   1:  PR[91,2] = PR[90,2] + -8.319;
   1:  PR[91,3] = PR[90,3] + 6.919;
   1:L PR[91] R[100]mm/sec CNT100;
   1:  PR[91,1] = PR[90,1] + 34.688;
   1:  PR[91,2] = PR[90,2] + -7.593;
   1:  PR[91,3] = PR[90,3] + 6.924;
   1:L PR[91] R[100]mm/sec CNT100;
   1:  PR[91,1] = PR[90,1] + 35.067;
   1:  PR[91,2] = PR[90,2] + -6.848;
   1:  PR[91,3] = PR[90,3] + 6.929;
   1:L PR[91] R[100]mm/sec CNT100;
   1:  PR[91,1] = PR[90,1] + 35.409;
   1:  PR[91,2] = PR[90,2] + -6.085;
   1:  PR[91,3] = PR[90,3] + 6.934;
   1:L PR[91] R[100]mm/sec CNT100;
   1:  PR[91,1] = PR[90,1] + 35.712;
   1:  PR[91,2] = PR[90,2] + -5.307;
   1:  PR[91,3] = PR[90,3] + 6.939;
   1:L PR[91] R[100]mm/sec CNT100;
   1:  PR[91,1] = PR[90,1] + 35.976;
   1:  PR[91,2] = PR[90,2] + -4.515;
   1:  PR[91,3] = PR[90,3] + 6.944;
   1:L PR[91] R[100]mm/sec CNT100;
   1:  PR[91,1] = PR[90,1] + 36.201;
   1:  PR[91,2] = PR[90,2] + -3.712;
   1:  PR[91,3] = PR[90,3] + 6.950;
   1:L PR[91] R[100]mm/sec CNT100;
   1:  PR[91,1] = PR[90,1] + 36.386;
   1:  PR[91,2] = PR[90,2] + -2.898;
   1:  PR[91,3] = PR[90,3] + 6.955;
   1:L PR[91] R[100]mm/sec CNT100;
   1:  PR[91,1] = PR[90,1] + 36.530;
   1:  PR[91,2] = PR[90,2] + -2.076;
   1:  PR[91,3] = PR[90,3] + 6.960;
   1:L PR[91] R[100]mm/sec CNT100;
   1:  PR[91,1] = PR[90,1] + 36.633;
   1:  PR[91,2] = PR[90,2] + -1.246;
   1:  PR[91,3] = PR[90,3] + 6.965;
   1:L PR[91] R[100]mm/sec CNT100;
   1:  PR[91,1] = PR[90,1] + 36.695;
   1:  PR[91,2] = PR[90,2] + -0.411;
   1:  PR[91,3] = PR[90,3] + 6.970;
   1:L PR[91] R[100]mm/sec CNT100;
   1:  PR[91,1] = PR[90,1] + 36.716;
   1:  PR[91,2] = PR[90,2] + 0.428;
   1:  PR[91,3] = PR[90,3] + 6.975;
   1:L PR[91] R[100]mm/sec CNT100;
   1:  PR[91,1] = PR[90,1] + 36.695;
   1:  PR[91,2] = PR[90,2] + 1.266;
   1:  PR[91,3] = PR[90,3] + 6.980;
   1:L PR[91] R[100]mm/sec CNT100;
   1:  PR[91,1] = PR[90,1] + 36.633;
   1:  PR[91,2] = PR[90,2] + 2.101;
   1:  PR[91,3] = PR[90,3] + 6.985;
   1:L PR[91] R[100]mm/sec CNT100;
   1:  PR[91,1] = PR[90,1] + 36.530;
   1:  PR[91,2] = PR[90,2] + 2.931;
   1:  PR[91,3] = PR[90,3] + 6.990;
   1:L PR[91] R[100]mm/sec CNT100;
   1:  PR[91,1] = PR[90,1] + 36.386;
   1:  PR[91,2] = PR[90,2] + 3.753;
   1:  PR[91,3] = PR[90,3] + 6.995;
   1:L PR[91] R[100]mm/sec CNT100;
   1:  PR[91,1] = PR[90,1] + 36.201;
   1:  PR[91,2] = PR[90,2] + 4.567;
   1:  PR[91,3] = PR[90,3] + 7.000;
   1:L PR[91] R[100]mm/sec CNT100;
   1:  PR[91,1] = PR[90,1] + 35.976;
   1:  PR[91,2] = PR[90,2] + 5.371;
   1:  PR[91,3] = PR[90,3] + 7.005;
   1:L PR[91] R[100]mm/sec CNT100;
   1:  PR[91,1] = PR[90,1] + 35.712;
   1:  PR[91,2] = PR[90,2] + 6.162;
   1:  PR[91,3] = PR[90,3] + 7.011;
   1:L PR[91] R[100]mm/sec CNT100;
   1:  PR[91,1] = PR[90,1] + 35.409;
   1:  PR[91,2] = PR[90,2] + 6.940;
   1:  PR[91,3] = PR[90,3] + 7.016;
   1:L PR[91] R[100]mm/sec CNT100;
   1:  PR[91,1] = PR[90,1] + 35.067;
   1:  PR[91,2] = PR[90,2] + 7.703;
   1:  PR[91,3] = PR[90,3] + 7.021;
   1:L PR[91] R[100]mm/sec CNT100;
   1:  PR[91,1] = PR[90,1] + 34.688;
   1:  PR[91,2] = PR[90,2] + 8.449;
   1:  PR[91,3] = PR[90,3] + 7.026;
   1:L PR[91] R[100]mm/sec CNT100;
   1:  PR[91,1] = PR[90,1] + 34.273;
   1:  PR[91,2] = PR[90,2] + 9.175;
   1:  PR[91,3] = PR[90,3] + 7.031;
   1:L PR[91] R[100]mm/sec CNT100;
   1:  PR[91,1] = PR[90,1] + 33.822;
   1:  PR[91,2] = PR[90,2] + 9.879;
   1:  PR[91,3] = PR[90,3] + 7.036;
   1:L PR[91] R[100]mm/sec CNT100;
   1:  PR[91,1] = PR[90,1] + 33.337;
   1:  PR[91,2] = PR[90,2] + 10.561;
   1:  PR[91,3] = PR[90,3] + 7.041;
   1:L PR[91] R[100]mm/sec CNT100;
   1:  PR[91,1] = PR[90,1] + 32.819;
   1:  PR[91,2] = PR[90,2] + 11.219;
   1:  PR[91,3] = PR[90,3] + 7.046;
   1:L PR[91] R[100]mm/sec CNT100;
   1:  PR[91,1] = PR[90,1] + 32.269;
   1:  PR[91,2] = PR[90,2] + 11.849;
   1:  PR[91,3] = PR[90,3] + 7.051;
   1:L PR[91] R[100]mm/sec CNT100;
   1:  PR[91,1] = PR[90,1] + 31.688;
   1:  PR[91,2] = PR[90,2] + 12.452;
   1:  PR[91,3] = PR[90,3] + 7.056;
   1:L PR[91] R[100]mm/sec CNT100;
   1:  PR[91,1] = PR[90,1] + 31.079;
   1:  PR[91,2] = PR[90,2] + 13.025;
   1:  PR[91,3] = PR[90,3] + 7.061;
   1:L PR[91] R[100]mm/sec CNT100;
   1:  PR[91,1] = PR[90,1] + 30.441;
   1:  PR[91,2] = PR[90,2] + 13.567;
   1:  PR[91,3] = PR[90,3] + 7.067;
   1:L PR[91] R[100]mm/sec CNT100;
   1:  PR[91,1] = PR[90,1] + 29.778;
   1:  PR[91,2] = PR[90,2] + 14.078;
   1:  PR[91,3] = PR[90,3] + 7.072;
   1:L PR[91] R[100]mm/sec CNT100;
   1:  PR[91,1] = PR[90,1] + 29.090;
   1:  PR[91,2] = PR[90,2] + 14.555;
   1:  PR[91,3] = PR[90,3] + 7.077;
   1:L PR[91] R[100]mm/sec CNT100;
   1:  PR[91,1] = PR[90,1] + 28.379;
   1:  PR[91,2] = PR[90,2] + 14.998;
   1:  PR[91,3] = PR[90,3] + 7.082;
   1:L PR[91] R[100]mm/sec CNT100;
   1:  PR[91,1] = PR[90,1] + 27.647;
   1:  PR[91,2] = PR[90,2] + 15.405;
   1:  PR[91,3] = PR[90,3] + 7.087;
   1:L PR[91] R[100]mm/sec CNT100;
   1:  PR[91,1] = PR[90,1] + 26.895;
   1:  PR[91,2] = PR[90,2] + 15.775;
   1:  PR[91,3] = PR[90,3] + 7.092;
   1:L PR[91] R[100]mm/sec CNT100;
   1:  PR[91,1] = PR[90,1] + 26.126;
   1:  PR[91,2] = PR[90,2] + 16.108;
   1:  PR[91,3] = PR[90,3] + 7.097;
   1:L PR[91] R[100]mm/sec CNT100;
   1:  PR[91,1] = PR[90,1] + 25.342;
   1:  PR[91,2] = PR[90,2] + 16.403;
   1:  PR[91,3] = PR[90,3] + 7.102;
   1:L PR[91] R[100]mm/sec CNT100;
   1:  PR[91,1] = PR[90,1] + 24.544;
   1:  PR[91,2] = PR[90,2] + 16.659;
   1:  PR[91,3] = PR[90,3] + 7.107;
   1:L PR[91] R[100]mm/sec CNT100;
   1:  PR[91,1] = PR[90,1] + 23.734;
   1:  PR[91,2] = PR[90,2] + 16.875;
   1:  PR[91,3] = PR[90,3] + 7.112;
   1:L PR[91] R[100]mm/sec CNT100;
   1:  PR[91,1] = PR[90,1] + 22.914;
   1:  PR[91,2] = PR[90,2] + 17.051;
   1:  PR[91,3] = PR[90,3] + 7.117;
   1:L PR[91] R[100]mm/sec CNT100;
   1:  PR[91,1] = PR[90,1] + 22.086;
   1:  PR[91,2] = PR[90,2] + 17.187;
   1:  PR[91,3] = PR[90,3] + 7.123;
   1:L PR[91] R[100]mm/sec CNT100;
   1:  PR[91,1] = PR[90,1] + 21.253;
   1:  PR[91,2] = PR[90,2] + 17.281;
   1:  PR[91,3] = PR[90,3] + 7.128;
   1:L PR[91] R[100]mm/sec CNT100;
   1:  PR[91,1] = PR[90,1] + 20.416;
   1:  PR[91,2] = PR[90,2] + 17.335;
   1:  PR[91,3] = PR[90,3] + 7.133;
   1:L PR[91] R[100]mm/sec CNT100;
   1:  PR[91,1] = PR[90,1] + 19.577;
   1:  PR[91,2] = PR[90,2] + 17.347;
   1:  PR[91,3] = PR[90,3] + 7.138;
   1:L PR[91] R[100]mm/sec CNT100;
   1:  PR[91,1] = PR[90,1] + 18.739;
   1:  PR[91,2] = PR[90,2] + 17.318;
   1:  PR[91,3] = PR[90,3] + 7.143;
   1:L PR[91] R[100]mm/sec CNT100;
   1:  PR[91,1] = PR[90,1] + 17.902;
   1:  PR[91,2] = PR[90,2] + 17.247;
   1:  PR[91,3] = PR[90,3] + 7.148;
   1:L PR[91] R[100]mm/sec CNT100;
   1:  PR[91,1] = PR[90,1] + 17.071;
   1:  PR[91,2] = PR[90,2] + 17.136;
   1:  PR[91,3] = PR[90,3] + 7.153;
   1:L PR[91] R[100]mm/sec CNT100;
   1:  PR[91,1] = PR[90,1] + 16.226;
   1:  PR[91,2] = PR[90,2] + 16.978;
   1:  PR[91,3] = PR[90,3] + 7.158;
   1:L PR[91] R[100]mm/sec CNT100;
   1:  PR[91,1] = PR[90,1] + 15.428;
   1:  PR[91,2] = PR[90,2] + 16.790;
   1:  PR[91,3] = PR[90,3] + 7.164;
   1:L PR[91] R[100]mm/sec CNT100;
   1:  PR[91,1] = PR[90,1] + 14.620;
   1:  PR[91,2] = PR[90,2] + 16.557;
   1:  PR[91,3] = PR[90,3] + 7.168;
   1:L PR[91] R[100]mm/sec CNT100;
   1:  PR[91,1] = PR[90,1] + 13.825;
   1:  PR[91,2] = PR[90,2] + 16.285;
   1:  PR[91,3] = PR[90,3] + 7.174;
   1:L PR[91] R[100]mm/sec CNT100;
   1:  PR[91,1] = PR[90,1] + 13.044;
   1:  PR[91,2] = PR[90,2] + 15.974;
   1:  PR[91,3] = PR[90,3] + 7.179;
   1:L PR[91] R[100]mm/sec CNT100;
   1:  PR[91,1] = PR[90,1] + 12.279;
   1:  PR[91,2] = PR[90,2] + 15.624;
   1:  PR[91,3] = PR[90,3] + 7.184;
   1:L PR[91] R[100]mm/sec CNT100;
   1:  PR[91,1] = PR[90,1] + 11.533;
   1:  PR[91,2] = PR[90,2] + 15.238;
   1:  PR[91,3] = PR[90,3] + 7.189;
   1:L PR[91] R[100]mm/sec CNT100;
   1:  PR[91,1] = PR[90,1] + 10.807;
   1:  PR[91,2] = PR[90,2] + 14.816;
   1:  PR[91,3] = PR[90,3] + 7.194;
   1:L PR[91] R[100]mm/sec CNT100;
   1:  PR[91,1] = PR[90,1] + 10.102;
   1:  PR[91,2] = PR[90,2] + 14.358;
   1:  PR[91,3] = PR[90,3] + 7.199;
   1:L PR[91] R[100]mm/sec CNT100;
   1:  PR[91,1] = PR[90,1] + 9.421;
   1:  PR[91,2] = PR[90,2] + 13.866;
   1:  PR[91,3] = PR[90,3] + 7.204;
   1:L PR[91] R[100]mm/sec CNT100;
   1:  PR[91,1] = PR[90,1] + 8.765;
   1:  PR[91,2] = PR[90,2] + 13.341;
   1:  PR[91,3] = PR[90,3] + 7.209;
   1:L PR[91] R[100]mm/sec CNT100;
   1:  PR[91,1] = PR[90,1] + 8.136;
   1:  PR[91,2] = PR[90,2] + 12.785;
   1:  PR[91,3] = PR[90,3] + 7.214;
   1:L PR[91] R[100]mm/sec CNT100;
   1:  PR[91,1] = PR[90,1] + 7.535;
   1:  PR[91,2] = PR[90,2] + 12.198;
   1:  PR[91,3] = PR[90,3] + 7.220;
   1:L PR[91] R[100]mm/sec CNT100;
   1:  PR[91,1] = PR[90,1] + 6.965;
   1:  PR[91,2] = PR[90,2] + 11.581;
   1:  PR[91,3] = PR[90,3] + 7.225;
   1:L PR[91] R[100]mm/sec CNT100;
   1:  PR[91,1] = PR[90,1] + 6.425;
   1:  PR[91,2] = PR[90,2] + 10.938;
   1:  PR[91,3] = PR[90,3] + 7.230;
   1:L PR[91] R[100]mm/sec CNT100;
   1:  PR[91,1] = PR[90,1] + 5.918;
   1:  PR[91,2] = PR[90,2] + 10.268;
   1:  PR[91,3] = PR[90,3] + 7.235;
   1:L PR[91] R[100]mm/sec CNT100;
   1:  PR[91,1] = PR[90,1] + 5.445;
   1:  PR[91,2] = PR[90,2] + 9.574;
   1:  PR[91,3] = PR[90,3] + 7.240;
   1:L PR[91] R[100]mm/sec CNT100;
   1:  PR[91,1] = PR[90,1] + 5.007;
   1:  PR[91,2] = PR[90,2] + 8.857;
   1:  PR[91,3] = PR[90,3] + 7.245;
   1:L PR[91] R[100]mm/sec CNT100;
   1:  PR[91,1] = PR[90,1] + 4.605;
   1:  PR[91,2] = PR[90,2] + 8.120;
   1:  PR[91,3] = PR[90,3] + 7.250;
   1:L PR[91] R[100]mm/sec CNT100;
   1:  PR[91,1] = PR[90,1] + 4.240;
   1:  PR[91,2] = PR[90,2] + 7.365;
   1:  PR[91,3] = PR[90,3] + 7.255;
   1:L PR[91] R[100]mm/sec CNT100;
   1:  PR[91,1] = PR[90,1] + 3.913;
   1:  PR[91,2] = PR[90,2] + 6.594;
   1:  PR[91,3] = PR[90,3] + 7.260;
   1:L PR[91] R[100]mm/sec CNT100;
   1:  PR[91,1] = PR[90,1] + 3.625;
   1:  PR[91,2] = PR[90,2] + 5.810;
   1:  PR[91,3] = PR[90,3] + 7.266;
   1:L PR[91] R[100]mm/sec CNT100;
   1:  PR[91,1] = PR[90,1] + 3.377;
   1:  PR[91,2] = PR[90,2] + 5.013;
   1:  PR[91,3] = PR[90,3] + 7.271;
   1:L PR[91] R[100]mm/sec CNT100;
   1:  PR[91,1] = PR[90,1] + 3.169;
   1:  PR[91,2] = PR[90,2] + 4.205;
   1:  PR[91,3] = PR[90,3] + 7.276;
   1:L PR[91] R[100]mm/sec CNT100;
   1:  PR[91,1] = PR[90,1] + 2.997;
   1:  PR[91,2] = PR[90,2] + 3.358;
   1:  PR[91,3] = PR[90,3] + 7.281;
   1:L PR[91] R[100]mm/sec CNT100;
   1:  PR[91,1] = PR[90,1] + 2.902;
   1:  PR[91,2] = PR[90,2] + 2.988;
   1:  PR[91,3] = PR[90,3] + 7.286;
   1:L PR[91] R[100]mm/sec CNT100;
   1:  PR[91,1] = PR[90,1] + 2.754;
   1:  PR[91,2] = PR[90,2] + 2.613;
   1:  PR[91,3] = PR[90,3] + 7.288;
   1:L PR[91] R[100]mm/sec CNT100;
   1:  PR[91,1] = PR[90,1] + 2.570;
   1:  PR[91,2] = PR[90,2] + 2.280;
   1:  PR[91,3] = PR[90,3] + 7.291;
   1:L PR[91] R[100]mm/sec CNT100;
   1:  PR[91,1] = PR[90,1] + 2.373;
   1:  PR[91,2] = PR[90,2] + 2.003;
   1:  PR[91,3] = PR[90,3] + 7.293;
   1:L PR[91] R[100]mm/sec CNT100;
   1:  PR[91,1] = PR[90,1] + 2.094;
   1:  PR[91,2] = PR[90,2] + 1.696;
   1:  PR[91,3] = PR[90,3] + 7.295;
   1:L PR[91] R[100]mm/sec CNT100;
   1:  PR[91,1] = PR[90,1] + 1.771;
   1:  PR[91,2] = PR[90,2] + 1.427;
   1:  PR[91,3] = PR[90,3] + 7.298;
   1:L PR[91] R[100]mm/sec CNT100;
   1:  PR[91,1] = PR[90,1] + 1.413;
   1:  PR[91,2] = PR[90,2] + 1.202;
   1:  PR[91,3] = PR[90,3] + 7.300;
   1:L PR[91] R[100]mm/sec CNT100;
   1:  PR[91,1] = PR[90,1] + 1.037;
   1:  PR[91,2] = PR[90,2] + 1.031;
   1:  PR[91,3] = PR[90,3] + 7.303;
   1:L PR[91] R[100]mm/sec CNT100;
   1:  PR[91,1] = PR[90,1] + 0.744;
   1:  PR[91,2] = PR[90,2] + 0.936;
   1:  PR[91,3] = PR[90,3] + 7.305;
   1:L PR[91] R[100]mm/sec CNT100;
   1:  PR[91,1] = PR[90,1] + 0.340;
   1:  PR[91,2] = PR[90,2] + 0.854;
   1:  PR[91,3] = PR[90,3] + 7.307;
   1:L PR[91] R[100]mm/sec CNT100;
   1:  PR[91,1] = PR[90,1] + -0.072;
   1:  PR[91,2] = PR[90,2] + 0.827;
   1:  PR[91,3] = PR[90,3] + 7.310;
   1:L PR[91] R[100]mm/sec CNT100;
   1:  PR[91,1] = PR[90,1] + -0.523;
   1:  PR[91,2] = PR[90,2] + 0.847;
   1:  PR[91,3] = PR[90,3] + 7.312;
   1:L PR[91] R[100]mm/sec CNT100;
   1:  PR[91,1] = PR[90,1] + -0.953;
   1:  PR[91,2] = PR[90,2] + 0.928;
   1:  PR[91,3] = PR[90,3] + 7.315;
   1:L PR[91] R[100]mm/sec CNT100;
   1:  PR[91,1] = PR[90,1] + -1.273;
   1:  PR[91,2] = PR[90,2] + 1.030;
   1:  PR[91,3] = PR[90,3] + 7.318;
   1:L PR[91] R[100]mm/sec CNT100;
   1:  PR[91,1] = PR[90,1] + -1.637;
   1:  PR[91,2] = PR[90,2] + 1.194;
   1:  PR[91,3] = PR[90,3] + 7.320;
   1:L PR[91] R[100]mm/sec CNT100;
   1:  PR[91,1] = PR[90,1] + -1.982;
   1:  PR[91,2] = PR[90,2] + 1.407;
   1:  PR[91,3] = PR[90,3] + 7.322;
   1:L PR[91] R[100]mm/sec CNT100;
   1:  PR[91,1] = PR[90,1] + -2.261;
   1:  PR[91,2] = PR[90,2] + 1.632;
   1:  PR[91,3] = PR[90,3] + 7.325;
   1:L PR[91] R[100]mm/sec CNT100;
   1:  PR[91,1] = PR[90,1] + -2.628;
   1:  PR[91,2] = PR[90,2] + 2.025;
   1:  PR[91,3] = PR[90,3] + 7.327;
   1:L PR[91] R[100]mm/sec CNT100;
   1:  PR[91,1] = PR[90,1] + -2.823;
   1:  PR[91,2] = PR[90,2] + 2.302;
   1:  PR[91,3] = PR[90,3] + 7.330;
   1:L PR[91] R[100]mm/sec CNT100;
   1:  PR[91,1] = PR[90,1] + -3.001;
   1:  PR[91,2] = PR[90,2] + 2.631;
   1:  PR[91,3] = PR[90,3] + 7.332;
   1:L PR[91] R[100]mm/sec CNT100;
   1:  PR[91,1] = PR[90,1] + -3.158;
   1:  PR[91,2] = PR[90,2] + 3.044;
   1:  PR[91,3] = PR[90,3] + 7.334;
   1:L PR[91] R[100]mm/sec CNT100;
   1:  PR[91,1] = PR[90,1] + -3.406;
   1:  PR[91,2] = PR[90,2] + 4.200;
   1:  PR[91,3] = PR[90,3] + 7.337;
   1:L PR[91] R[100]mm/sec CNT100;
   1:  PR[91,1] = PR[90,1] + -3.615;
   1:  PR[91,2] = PR[90,2] + 5.011;
   1:  PR[91,3] = PR[90,3] + 7.344;
   1:L PR[91] R[100]mm/sec CNT100;
   1:  PR[91,1] = PR[90,1] + -3.864;
   1:  PR[91,2] = PR[90,2] + 5.809;
   1:  PR[91,3] = PR[90,3] + 7.349;
   1:L PR[91] R[100]mm/sec CNT100;
   1:  PR[91,1] = PR[90,1] + -4.152;
   1:  PR[91,2] = PR[90,2] + 6.594;
   1:  PR[91,3] = PR[90,3] + 7.354;
   1:L PR[91] R[100]mm/sec CNT100;
   1:  PR[91,1] = PR[90,1] + -4.479;
   1:  PR[91,2] = PR[90,2] + 7.366;
   1:  PR[91,3] = PR[90,3] + 7.360;
   1:L PR[91] R[100]mm/sec CNT100;
   1:  PR[91,1] = PR[90,1] + -4.844;
   1:  PR[91,2] = PR[90,2] + 8.122;
   1:  PR[91,3] = PR[90,3] + 7.365;
   1:L PR[91] R[100]mm/sec CNT100;
   1:  PR[91,1] = PR[90,1] + -5.246;
   1:  PR[91,2] = PR[90,2] + 8.859;
   1:  PR[91,3] = PR[90,3] + 7.370;
   1:L PR[91] R[100]mm/sec CNT100;
   1:  PR[91,1] = PR[90,1] + -5.684;
   1:  PR[91,2] = PR[90,2] + 9.576;
   1:  PR[91,3] = PR[90,3] + 7.375;
   1:L PR[91] R[100]mm/sec CNT100;
   1:  PR[91,1] = PR[90,1] + -6.157;
   1:  PR[91,2] = PR[90,2] + 10.270;
   1:  PR[91,3] = PR[90,3] + 7.380;
   1:L PR[91] R[100]mm/sec CNT100;
   1:  PR[91,1] = PR[90,1] + -6.664;
   1:  PR[91,2] = PR[90,2] + 10.939;
   1:  PR[91,3] = PR[90,3] + 7.385;
   1:L PR[91] R[100]mm/sec CNT100;
   1:  PR[91,1] = PR[90,1] + -7.204;
   1:  PR[91,2] = PR[90,2] + 11.583;
   1:  PR[91,3] = PR[90,3] + 7.390;
   1:L PR[91] R[100]mm/sec CNT100;
   1:  PR[91,1] = PR[90,1] + -7.775;
   1:  PR[91,2] = PR[90,2] + 12.198;
   1:  PR[91,3] = PR[90,3] + 7.395;
   1:L PR[91] R[100]mm/sec CNT100;
   1:  PR[91,1] = PR[90,1] + -8.375;
   1:  PR[91,2] = PR[90,2] + 12.785;
   1:  PR[91,3] = PR[90,3] + 7.400;
   1:L PR[91] R[100]mm/sec CNT100;
   1:  PR[91,1] = PR[90,1] + -9.004;
   1:  PR[91,2] = PR[90,2] + 13.341;
   1:  PR[91,3] = PR[90,3] + 7.405;
   1:L PR[91] R[100]mm/sec CNT100;
   1:  PR[91,1] = PR[90,1] + -9.660;
   1:  PR[91,2] = PR[90,2] + 13.866;
   1:  PR[91,3] = PR[90,3] + 7.411;
   1:L PR[91] R[100]mm/sec CNT100;
   1:  PR[91,1] = PR[90,1] + -10.341;
   1:  PR[91,2] = PR[90,2] + 14.358;
   1:  PR[91,3] = PR[90,3] + 7.416;
   1:L PR[91] R[100]mm/sec CNT100;
   1:  PR[91,1] = PR[90,1] + -11.046;
   1:  PR[91,2] = PR[90,2] + 14.816;
   1:  PR[91,3] = PR[90,3] + 7.421;
   1:L PR[91] R[100]mm/sec CNT100;
   1:  PR[91,1] = PR[90,1] + -11.772;
   1:  PR[91,2] = PR[90,2] + 15.238;
   1:  PR[91,3] = PR[90,3] + 7.426;
   1:L PR[91] R[100]mm/sec CNT100;
   1:  PR[91,1] = PR[90,1] + -12.519;
   1:  PR[91,2] = PR[90,2] + 15.625;
   1:  PR[91,3] = PR[90,3] + 7.431;
   1:L PR[91] R[100]mm/sec CNT100;
   1:  PR[91,1] = PR[90,1] + -13.283;
   1:  PR[91,2] = PR[90,2] + 15.974;
   1:  PR[91,3] = PR[90,3] + 7.436;
   1:L PR[91] R[100]mm/sec CNT100;
   1:  PR[91,1] = PR[90,1] + -14.064;
   1:  PR[91,2] = PR[90,2] + 16.285;
   1:  PR[91,3] = PR[90,3] + 7.441;
   1:L PR[91] R[100]mm/sec CNT100;
   1:  PR[91,1] = PR[90,1] + -14.859;
   1:  PR[91,2] = PR[90,2] + 16.557;
   1:  PR[91,3] = PR[90,3] + 7.446;
   1:L PR[91] R[100]mm/sec CNT100;
   1:  PR[91,1] = PR[90,1] + -15.678;
   1:  PR[91,2] = PR[90,2] + 16.793;
   1:  PR[91,3] = PR[90,3] + 7.451;
   1:L PR[91] R[100]mm/sec CNT100;
   1:  PR[91,1] = PR[90,1] + -16.484;
   1:  PR[91,2] = PR[90,2] + 16.983;
   1:  PR[91,3] = PR[90,3] + 7.457;
   1:L PR[91] R[100]mm/sec CNT100;
   1:  PR[91,1] = PR[90,1] + -17.310;
   1:  PR[91,2] = PR[90,2] + 17.136;
   1:  PR[91,3] = PR[90,3] + 7.462;
   1:L PR[91] R[100]mm/sec CNT100;
   1:  PR[91,1] = PR[90,1] + -18.141;
   1:  PR[91,2] = PR[90,2] + 17.247;
   1:  PR[91,3] = PR[90,3] + 7.467;
   1:L PR[91] R[100]mm/sec CNT100;
   1:  PR[91,1] = PR[90,1] + -18.978;
   1:  PR[91,2] = PR[90,2] + 17.318;
   1:  PR[91,3] = PR[90,3] + 7.472;
   1:L PR[91] R[100]mm/sec CNT100;
   1:  PR[91,1] = PR[90,1] + -19.816;
   1:  PR[91,2] = PR[90,2] + 17.347;
   1:  PR[91,3] = PR[90,3] + 7.477;
   1:L PR[91] R[100]mm/sec CNT100;
   1:  PR[91,1] = PR[90,1] + -20.655;
   1:  PR[91,2] = PR[90,2] + 17.335;
   1:  PR[91,3] = PR[90,3] + 7.482;
   1:L PR[91] R[100]mm/sec CNT100;
   1:  PR[91,1] = PR[90,1] + -21.492;
   1:  PR[91,2] = PR[90,2] + 17.281;
   1:  PR[91,3] = PR[90,3] + 7.487;
   1:L PR[91] R[100]mm/sec CNT100;
   1:  PR[91,1] = PR[90,1] + -22.325;
   1:  PR[91,2] = PR[90,2] + 17.187;
   1:  PR[91,3] = PR[90,3] + 7.492;
   1:L PR[91] R[100]mm/sec CNT100;
   1:  PR[91,1] = PR[90,1] + -23.153;
   1:  PR[91,2] = PR[90,2] + 17.051;
   1:  PR[91,3] = PR[90,3] + 7.497;
   1:L PR[91] R[100]mm/sec CNT100;
   1:  PR[91,1] = PR[90,1] + -23.973;
   1:  PR[91,2] = PR[90,2] + 16.875;
   1:  PR[91,3] = PR[90,3] + 7.503;
   1:L PR[91] R[100]mm/sec CNT100;
   1:  PR[91,1] = PR[90,1] + -24.783;
   1:  PR[91,2] = PR[90,2] + 16.659;
   1:  PR[91,3] = PR[90,3] + 7.508;
   1:L PR[91] R[100]mm/sec CNT100;
   1:  PR[91,1] = PR[90,1] + -25.581;
   1:  PR[91,2] = PR[90,2] + 16.403;
   1:  PR[91,3] = PR[90,3] + 7.513;
   1:L PR[91] R[100]mm/sec CNT100;
   1:  PR[91,1] = PR[90,1] + -26.365;
   1:  PR[91,2] = PR[90,2] + 16.108;
   1:  PR[91,3] = PR[90,3] + 7.518;
   1:L PR[91] R[100]mm/sec CNT100;
   1:  PR[91,1] = PR[90,1] + -27.134;
   1:  PR[91,2] = PR[90,2] + 15.775;
   1:  PR[91,3] = PR[90,3] + 7.523;
   1:L PR[91] R[100]mm/sec CNT100;
   1:  PR[91,1] = PR[90,1] + -27.885;
   1:  PR[91,2] = PR[90,2] + 15.404;
   1:  PR[91,3] = PR[90,3] + 7.528;
   1:L PR[91] R[100]mm/sec CNT100;
   1:  PR[91,1] = PR[90,1] + -28.617;
   1:  PR[91,2] = PR[90,2] + 14.997;
   1:  PR[91,3] = PR[90,3] + 7.533;
   1:L PR[91] R[100]mm/sec CNT100;
   1:  PR[91,1] = PR[90,1] + -29.328;
   1:  PR[91,2] = PR[90,2] + 14.555;
   1:  PR[91,3] = PR[90,3] + 7.538;
   1:L PR[91] R[100]mm/sec CNT100;
   1:  PR[91,1] = PR[90,1] + -30.016;
   1:  PR[91,2] = PR[90,2] + 14.077;
   1:  PR[91,3] = PR[90,3] + 7.543;
   1:L PR[91] R[100]mm/sec CNT100;
   1:  PR[91,1] = PR[90,1] + -30.680;
   1:  PR[91,2] = PR[90,2] + 13.567;
   1:  PR[91,3] = PR[90,3] + 7.548;
   1:L PR[91] R[100]mm/sec CNT100;
   1:  PR[91,1] = PR[90,1] + -31.317;
   1:  PR[91,2] = PR[90,2] + 13.025;
   1:  PR[91,3] = PR[90,3] + 7.553;
   1:L PR[91] R[100]mm/sec CNT100;
   1:  PR[91,1] = PR[90,1] + -31.927;
   1:  PR[91,2] = PR[90,2] + 12.451;
   1:  PR[91,3] = PR[90,3] + 7.559;
   1:L PR[91] R[100]mm/sec CNT100;
   1:  PR[91,1] = PR[90,1] + -32.508;
   1:  PR[91,2] = PR[90,2] + 11.849;
   1:  PR[91,3] = PR[90,3] + 7.564;
   1:L PR[91] R[100]mm/sec CNT100;
   1:  PR[91,1] = PR[90,1] + -33.058;
   1:  PR[91,2] = PR[90,2] + 11.219;
   1:  PR[91,3] = PR[90,3] + 7.569;
   1:L PR[91] R[100]mm/sec CNT100;
   1:  PR[91,1] = PR[90,1] + -33.576;
   1:  PR[91,2] = PR[90,2] + 10.562;
   1:  PR[91,3] = PR[90,3] + 7.574;
   1:L PR[91] R[100]mm/sec CNT100;
   1:  PR[91,1] = PR[90,1] + -34.061;
   1:  PR[91,2] = PR[90,2] + 9.880;
   1:  PR[91,3] = PR[90,3] + 7.579;
   1:L PR[91] R[100]mm/sec CNT100;
   1:  PR[91,1] = PR[90,1] + -34.512;
   1:  PR[91,2] = PR[90,2] + 9.175;
   1:  PR[91,3] = PR[90,3] + 7.584;
   1:L PR[91] R[100]mm/sec CNT100;
   1:  PR[91,1] = PR[90,1] + -34.927;
   1:  PR[91,2] = PR[90,2] + 8.449;
   1:  PR[91,3] = PR[90,3] + 7.589;
   1:L PR[91] R[100]mm/sec CNT100;
   1:  PR[91,1] = PR[90,1] + -35.306;
   1:  PR[91,2] = PR[90,2] + 7.703;
   1:  PR[91,3] = PR[90,3] + 7.594;
   1:L PR[91] R[100]mm/sec CNT100;
   1:  PR[91,1] = PR[90,1] + -35.647;
   1:  PR[91,2] = PR[90,2] + 6.940;
   1:  PR[91,3] = PR[90,3] + 7.599;
   1:L PR[91] R[100]mm/sec CNT100;
   1:  PR[91,1] = PR[90,1] + -35.950;
   1:  PR[91,2] = PR[90,2] + 6.161;
   1:  PR[91,3] = PR[90,3] + 7.604;
   1:L PR[91] R[100]mm/sec CNT100;
   1:  PR[91,1] = PR[90,1] + -36.215;
   1:  PR[91,2] = PR[90,2] + 5.370;
   1:  PR[91,3] = PR[90,3] + 7.609;
   1:L PR[91] R[100]mm/sec CNT100;
   1:  PR[91,1] = PR[90,1] + -36.440;
   1:  PR[91,2] = PR[90,2] + 4.566;
   1:  PR[91,3] = PR[90,3] + 7.615;
   1:L PR[91] R[100]mm/sec CNT100;
   1:  PR[91,1] = PR[90,1] + -36.624;
   1:  PR[91,2] = PR[90,2] + 3.752;
   1:  PR[91,3] = PR[90,3] + 7.620;
   1:L PR[91] R[100]mm/sec CNT100;
   1:  PR[91,1] = PR[90,1] + -36.768;
   1:  PR[91,2] = PR[90,2] + 2.930;
   1:  PR[91,3] = PR[90,3] + 7.625;
   1:L PR[91] R[100]mm/sec CNT100;
   1:  PR[91,1] = PR[90,1] + -36.871;
   1:  PR[91,2] = PR[90,2] + 2.101;
   1:  PR[91,3] = PR[90,3] + 7.630;
   1:L PR[91] R[100]mm/sec CNT100;
   1:  PR[91,1] = PR[90,1] + -36.933;
   1:  PR[91,2] = PR[90,2] + 1.266;
   1:  PR[91,3] = PR[90,3] + 7.635;
   1:L PR[91] R[100]mm/sec CNT100;
   1:  PR[91,1] = PR[90,1] + -36.954;
   1:  PR[91,2] = PR[90,2] + 0.428;
   1:  PR[91,3] = PR[90,3] + 7.640;
   1:L PR[91] R[100]mm/sec CNT100;
   1:  PR[91,1] = PR[90,1] + -36.933;
   1:  PR[91,2] = PR[90,2] + -0.411;
   1:  PR[91,3] = PR[90,3] + 7.645;
   1:L PR[91] R[100]mm/sec CNT100;
   1:  PR[91,1] = PR[90,1] + -36.871;
   1:  PR[91,2] = PR[90,2] + -1.246;
   1:  PR[91,3] = PR[90,3] + 7.650;
   1:L PR[91] R[100]mm/sec CNT100;
   1:  PR[91,1] = PR[90,1] + -36.768;
   1:  PR[91,2] = PR[90,2] + -2.075;
   1:  PR[91,3] = PR[90,3] + 7.655;
   1:L PR[91] R[100]mm/sec CNT100;
   1:  PR[91,1] = PR[90,1] + -36.624;
   1:  PR[91,2] = PR[90,2] + -2.897;
   1:  PR[91,3] = PR[90,3] + 7.660;
   1:L PR[91] R[100]mm/sec CNT100;
   1:  PR[91,1] = PR[90,1] + -36.440;
   1:  PR[91,2] = PR[90,2] + -3.711;
   1:  PR[91,3] = PR[90,3] + 7.665;
   1:L PR[91] R[100]mm/sec CNT100;
   1:  PR[91,1] = PR[90,1] + -36.215;
   1:  PR[91,2] = PR[90,2] + -4.514;
   1:  PR[91,3] = PR[90,3] + 7.670;
   1:L PR[91] R[100]mm/sec CNT100;
   1:  PR[91,1] = PR[90,1] + -35.950;
   1:  PR[91,2] = PR[90,2] + -5.306;
   1:  PR[91,3] = PR[90,3] + 7.676;
   1:L PR[91] R[100]mm/sec CNT100;
   1:  PR[91,1] = PR[90,1] + -35.647;
   1:  PR[91,2] = PR[90,2] + -6.085;
   1:  PR[91,3] = PR[90,3] + 7.681;
   1:L PR[91] R[100]mm/sec CNT100;
   1:  PR[91,1] = PR[90,1] + -35.306;
   1:  PR[91,2] = PR[90,2] + -6.848;
   1:  PR[91,3] = PR[90,3] + 7.686;
   1:L PR[91] R[100]mm/sec CNT100;
   1:  PR[91,1] = PR[90,1] + -34.927;
   1:  PR[91,2] = PR[90,2] + -7.594;
   1:  PR[91,3] = PR[90,3] + 7.691;
   1:L PR[91] R[100]mm/sec CNT100;
   1:  PR[91,1] = PR[90,1] + -34.512;
   1:  PR[91,2] = PR[90,2] + -8.320;
   1:  PR[91,3] = PR[90,3] + 7.696;
   1:L PR[91] R[100]mm/sec CNT100;
   1:  PR[91,1] = PR[90,1] + -34.061;
   1:  PR[91,2] = PR[90,2] + -9.025;
   1:  PR[91,3] = PR[90,3] + 7.701;
   1:L PR[91] R[100]mm/sec CNT100;
   1:  PR[91,1] = PR[90,1] + -33.576;
   1:  PR[91,2] = PR[90,2] + -9.706;
   1:  PR[91,3] = PR[90,3] + 7.706;
   1:L PR[91] R[100]mm/sec CNT100;
   1:  PR[91,1] = PR[90,1] + -33.058;
   1:  PR[91,2] = PR[90,2] + -10.363;
   1:  PR[91,3] = PR[90,3] + 7.711;
   1:L PR[91] R[100]mm/sec CNT100;
   1:  PR[91,1] = PR[90,1] + -32.508;
   1:  PR[91,2] = PR[90,2] + -10.994;
   1:  PR[91,3] = PR[90,3] + 7.716;
   1:L PR[91] R[100]mm/sec CNT100;
   1:  PR[91,1] = PR[90,1] + -31.927;
   1:  PR[91,2] = PR[90,2] + -11.596;
   1:  PR[91,3] = PR[90,3] + 7.721;
   1:L PR[91] R[100]mm/sec CNT100;
   1:  PR[91,1] = PR[90,1] + -31.317;
   1:  PR[91,2] = PR[90,2] + -12.170;
   1:  PR[91,3] = PR[90,3] + 7.726;
   1:L PR[91] R[100]mm/sec CNT100;
   1:  PR[91,1] = PR[90,1] + -30.680;
   1:  PR[91,2] = PR[90,2] + -12.712;
   1:  PR[91,3] = PR[90,3] + 7.731;
   1:L PR[91] R[100]mm/sec CNT100;
   1:  PR[91,1] = PR[90,1] + -30.016;
   1:  PR[91,2] = PR[90,2] + -13.222;
   1:  PR[91,3] = PR[90,3] + 7.737;
   1:L PR[91] R[100]mm/sec CNT100;
   1:  PR[91,1] = PR[90,1] + -29.328;
   1:  PR[91,2] = PR[90,2] + -13.699;
   1:  PR[91,3] = PR[90,3] + 7.742;
   1:L PR[91] R[100]mm/sec CNT100;
   1:  PR[91,1] = PR[90,1] + -28.617;
   1:  PR[91,2] = PR[90,2] + -14.142;
   1:  PR[91,3] = PR[90,3] + 7.747;
   1:L PR[91] R[100]mm/sec CNT100;
   1:  PR[91,1] = PR[90,1] + -27.885;
   1:  PR[91,2] = PR[90,2] + -14.549;
   1:  PR[91,3] = PR[90,3] + 7.752;
   1:L PR[91] R[100]mm/sec CNT100;
   1:  PR[91,1] = PR[90,1] + -27.134;
   1:  PR[91,2] = PR[90,2] + -14.920;
   1:  PR[91,3] = PR[90,3] + 7.757;
   1:L PR[91] R[100]mm/sec CNT100;
   1:  PR[91,1] = PR[90,1] + -26.365;
   1:  PR[91,2] = PR[90,2] + -15.253;
   1:  PR[91,3] = PR[90,3] + 7.762;
   1:L PR[91] R[100]mm/sec CNT100;
   1:  PR[91,1] = PR[90,1] + -25.581;
   1:  PR[91,2] = PR[90,2] + -15.548;
   1:  PR[91,3] = PR[90,3] + 7.767;
   1:L PR[91] R[100]mm/sec CNT100;
   1:  PR[91,1] = PR[90,1] + -24.782;
   1:  PR[91,2] = PR[90,2] + -15.804;
   1:  PR[91,3] = PR[90,3] + 7.772;
   1:L PR[91] R[100]mm/sec CNT100;
   1:  PR[91,1] = PR[90,1] + -23.973;
   1:  PR[91,2] = PR[90,2] + -16.020;
   1:  PR[91,3] = PR[90,3] + 7.777;
   1:L PR[91] R[100]mm/sec CNT100;
   1:  PR[91,1] = PR[90,1] + -23.153;
   1:  PR[91,2] = PR[90,2] + -16.196;
   1:  PR[91,3] = PR[90,3] + 7.782;
   1:L PR[91] R[100]mm/sec CNT100;
   1:  PR[91,1] = PR[90,1] + -22.325;
   1:  PR[91,2] = PR[90,2] + -16.332;
   1:  PR[91,3] = PR[90,3] + 7.788;
   1:L PR[91] R[100]mm/sec CNT100;
   1:  PR[91,1] = PR[90,1] + -21.492;
   1:  PR[91,2] = PR[90,2] + -16.426;
   1:  PR[91,3] = PR[90,3] + 7.793;
   1:L PR[91] R[100]mm/sec CNT100;
   1:  PR[91,1] = PR[90,1] + -20.655;
   1:  PR[91,2] = PR[90,2] + -16.480;
   1:  PR[91,3] = PR[90,3] + 7.798;
   1:L PR[91] R[100]mm/sec CNT100;
   1:  PR[91,1] = PR[90,1] + -19.816;
   1:  PR[91,2] = PR[90,2] + -16.492;
   1:  PR[91,3] = PR[90,3] + 7.803;
   1:L PR[91] R[100]mm/sec CNT100;
   1:  PR[91,1] = PR[90,1] + -18.978;
   1:  PR[91,2] = PR[90,2] + -16.463;
   1:  PR[91,3] = PR[90,3] + 7.808;
   1:L PR[91] R[100]mm/sec CNT100;
   1:  PR[91,1] = PR[90,1] + -18.141;
   1:  PR[91,2] = PR[90,2] + -16.392;
   1:  PR[91,3] = PR[90,3] + 7.813;
   1:L PR[91] R[100]mm/sec CNT100;
   1:  PR[91,1] = PR[90,1] + -17.310;
   1:  PR[91,2] = PR[90,2] + -16.280;
   1:  PR[91,3] = PR[90,3] + 7.818;
   1:L PR[91] R[100]mm/sec CNT100;
   1:  PR[91,1] = PR[90,1] + -16.484;
   1:  PR[91,2] = PR[90,2] + -16.128;
   1:  PR[91,3] = PR[90,3] + 7.823;
   1:L PR[91] R[100]mm/sec CNT100;
   1:  PR[91,1] = PR[90,1] + -15.667;
   1:  PR[91,2] = PR[90,2] + -15.935;
   1:  PR[91,3] = PR[90,3] + 7.828;
   1:L PR[91] R[100]mm/sec CNT100;
   1:  PR[91,1] = PR[90,1] + -14.859;
   1:  PR[91,2] = PR[90,2] + -15.702;
   1:  PR[91,3] = PR[90,3] + 7.833;
   1:L PR[91] R[100]mm/sec CNT100;
   1:  PR[91,1] = PR[90,1] + -14.064;
   1:  PR[91,2] = PR[90,2] + -15.430;
   1:  PR[91,3] = PR[90,3] + 7.839;
   1:L PR[91] R[100]mm/sec CNT100;
   1:  PR[91,1] = PR[90,1] + -13.283;
   1:  PR[91,2] = PR[90,2] + -15.119;
   1:  PR[91,3] = PR[90,3] + 7.844;
   1:L PR[91] R[100]mm/sec CNT100;
   1:  PR[91,1] = PR[90,1] + -12.519;
   1:  PR[91,2] = PR[90,2] + -14.770;
   1:  PR[91,3] = PR[90,3] + 7.849;
   1:L PR[91] R[100]mm/sec CNT100;
   1:  PR[91,1] = PR[90,1] + -11.772;
   1:  PR[91,2] = PR[90,2] + -14.383;
   1:  PR[91,3] = PR[90,3] + 7.854;
   1:L PR[91] R[100]mm/sec CNT100;
   1:  PR[91,1] = PR[90,1] + -11.046;
   1:  PR[91,2] = PR[90,2] + -13.961;
   1:  PR[91,3] = PR[90,3] + 7.859;
   1:L PR[91] R[100]mm/sec CNT100;
   1:  PR[91,1] = PR[90,1] + -10.341;
   1:  PR[91,2] = PR[90,2] + -13.503;
   1:  PR[91,3] = PR[90,3] + 7.864;
   1:L PR[91] R[100]mm/sec CNT100;
   1:  PR[91,1] = PR[90,1] + -9.660;
   1:  PR[91,2] = PR[90,2] + -13.011;
   1:  PR[91,3] = PR[90,3] + 7.869;
   1:L PR[91] R[100]mm/sec CNT100;
   1:  PR[91,1] = PR[90,1] + -9.004;
   1:  PR[91,2] = PR[90,2] + -12.486;
   1:  PR[91,3] = PR[90,3] + 7.874;
   1:L PR[91] R[100]mm/sec CNT100;
   1:  PR[91,1] = PR[90,1] + -8.375;
   1:  PR[91,2] = PR[90,2] + -11.930;
   1:  PR[91,3] = PR[90,3] + 7.879;
   1:L PR[91] R[100]mm/sec CNT100;
   1:  PR[91,1] = PR[90,1] + -7.775;
   1:  PR[91,2] = PR[90,2] + -11.343;
   1:  PR[91,3] = PR[90,3] + 7.885;
   1:L PR[91] R[100]mm/sec CNT100;
   1:  PR[91,1] = PR[90,1] + -7.204;
   1:  PR[91,2] = PR[90,2] + -10.728;
   1:  PR[91,3] = PR[90,3] + 7.890;
   1:L PR[91] R[100]mm/sec CNT100;
   1:  PR[91,1] = PR[90,1] + -6.664;
   1:  PR[91,2] = PR[90,2] + -10.084;
   1:  PR[91,3] = PR[90,3] + 7.895;
   1:L PR[91] R[100]mm/sec CNT100;
   1:  PR[91,1] = PR[90,1] + -6.157;
   1:  PR[91,2] = PR[90,2] + -9.415;
   1:  PR[91,3] = PR[90,3] + 7.900;
   1:L PR[91] R[100]mm/sec CNT100;
   1:  PR[91,1] = PR[90,1] + -5.684;
   1:  PR[91,2] = PR[90,2] + -8.721;
   1:  PR[91,3] = PR[90,3] + 7.905;
   1:L PR[91] R[100]mm/sec CNT100;
   1:  PR[91,1] = PR[90,1] + -5.246;
   1:  PR[91,2] = PR[90,2] + -8.004;
   1:  PR[91,3] = PR[90,3] + 7.910;
   1:L PR[91] R[100]mm/sec CNT100;
   1:  PR[91,1] = PR[90,1] + -4.844;
   1:  PR[91,2] = PR[90,2] + -7.267;
   1:  PR[91,3] = PR[90,3] + 7.915;
   1:L PR[91] R[100]mm/sec CNT100;
   1:  PR[91,1] = PR[90,1] + -4.479;
   1:  PR[91,2] = PR[90,2] + -6.511;
   1:  PR[91,3] = PR[90,3] + 7.920;
   1:L PR[91] R[100]mm/sec CNT100;
   1:  PR[91,1] = PR[90,1] + -4.152;
   1:  PR[91,2] = PR[90,2] + -5.739;
   1:  PR[91,3] = PR[90,3] + 7.925;
   1:L PR[91] R[100]mm/sec CNT100;
   1:  PR[91,1] = PR[90,1] + -3.864;
   1:  PR[91,2] = PR[90,2] + -4.954;
   1:  PR[91,3] = PR[90,3] + 7.931;
   1:L PR[91] R[100]mm/sec CNT100;
   1:  PR[91,1] = PR[90,1] + -3.615;
   1:  PR[91,2] = PR[90,2] + -4.156;
   1:  PR[91,3] = PR[90,3] + 7.936;
   1:L PR[91] R[100]mm/sec CNT100;
   1:  PR[91,1] = PR[90,1] + -3.407;
   1:  PR[91,2] = PR[90,2] + -3.349;
   1:  PR[91,3] = PR[90,3] + 7.941;
   1:L PR[91] R[100]mm/sec CNT100;
   1:  PR[91,1] = PR[90,1] + -3.236;
   1:  PR[91,2] = PR[90,2] + -2.502;
   1:  PR[91,3] = PR[90,3] + 7.946;
   1:L PR[91] R[100]mm/sec CNT100;
   1:  PR[91,1] = PR[90,1] + -3.140;
   1:  PR[91,2] = PR[90,2] + -2.132;
   1:  PR[91,3] = PR[90,3] + 7.951;
   1:L PR[91] R[100]mm/sec CNT100;
   1:  PR[91,1] = PR[90,1] + -2.992;
   1:  PR[91,2] = PR[90,2] + -1.757;
   1:  PR[91,3] = PR[90,3] + 7.953;
   1:L PR[91] R[100]mm/sec CNT100;
   1:  PR[91,1] = PR[90,1] + -2.807;
   1:  PR[91,2] = PR[90,2] + -1.421;
   1:  PR[91,3] = PR[90,3] + 7.956;
   1:L PR[91] R[100]mm/sec CNT100;
   1:  PR[91,1] = PR[90,1] + -2.567;
   1:  PR[91,2] = PR[90,2] + -1.093;
   1:  PR[91,3] = PR[90,3] + 7.958;
   1:L PR[91] R[100]mm/sec CNT100;
   1:  PR[91,1] = PR[90,1] + -2.301;
   1:  PR[91,2] = PR[90,2] + -0.812;
   1:  PR[91,3] = PR[90,3] + 7.961;
   1:L PR[91] R[100]mm/sec CNT100;
   1:  PR[91,1] = PR[90,1] + -2.011;
   1:  PR[91,2] = PR[90,2] + -0.573;
   1:  PR[91,3] = PR[90,3] + 7.963;
   1:L PR[91] R[100]mm/sec CNT100;
   1:  PR[91,1] = PR[90,1] + -1.740;
   1:  PR[91,2] = PR[90,2] + -0.397;
   1:  PR[91,3] = PR[90,3] + 7.965;
   1:L PR[91] R[100]mm/sec CNT100;
   1:  PR[91,1] = PR[90,1] + -1.380;
   1:  PR[91,2] = PR[90,2] + -0.217;
   1:  PR[91,3] = PR[90,3] + 7.967;
   1:L PR[91] R[100]mm/sec CNT100;
   1:  PR[91,1] = PR[90,1] + -0.988;
   1:  PR[91,2] = PR[90,2] + -0.082;
   1:  PR[91,3] = PR[90,3] + 7.970;
   1:L PR[91] R[100]mm/sec CNT100;
   1:  PR[91,1] = PR[90,1] + -0.579;
   1:  PR[91,2] = PR[90,2] + 0.001;
   1:  PR[91,3] = PR[90,3] + 7.972;
   1:L PR[91] R[100]mm/sec CNT100;
   1:  PR[91,1] = PR[90,1] + -0.167;
   1:  PR[91,2] = PR[90,2] + 0.028;
   1:  PR[91,3] = PR[90,3] + 7.975;
   1:L PR[91] R[100]mm/sec CNT100;
   1:  PR[91,1] = PR[90,1] + 0.284;
   1:  PR[91,2] = PR[90,2] + 0.008;
   1:  PR[91,3] = PR[90,3] + 7.977;
   1:L PR[91] R[100]mm/sec CNT100;
   1:  PR[91] = PR[90];
   1:  PR[91,1] = PR[90,1] + 0.988;
   1:  PR[91,2] = PR[90,2] + -0.431;
   1:  PR[91,3] = PR[90,3] + 9.310;
   1:L PR[91] R[100]mm/sec CNT100;
   1:  PR[91,1] = PR[90,1] + 1.508;
   1:  PR[91,2] = PR[90,2] + -0.717;
   1:  PR[91,3] = PR[90,3] + 7.984;
   1:L PR[91] R[100]mm/sec CNT100;
   1:  PR[91,1] = PR[90,1] + 1.978;
   1:  PR[91,2] = PR[90,2] + -1.118;
   1:  PR[91,3] = PR[90,3] + 7.987;
   1:L PR[91] R[100]mm/sec CNT100;
   1:  PR[91,1] = PR[90,1] + 2.298;
   1:  PR[91,2] = PR[90,2] + -1.539;
   1:  PR[91,3] = PR[90,3] + 7.991;
   1:L PR[91] R[100]mm/sec CNT100;
   1:  PR[91,1] = PR[90,1] + 2.452;
   1:  PR[91,2] = PR[90,2] + -1.800;
   1:  PR[91,3] = PR[90,3] + 7.994;
   1:L PR[91] R[100]mm/sec CNT100;
   1:  PR[91,1] = PR[90,1] + 2.588;
   1:  PR[91,2] = PR[90,2] + -2.085;
   1:  PR[91,3] = PR[90,3] + 7.996;
   1:L PR[91] R[100]mm/sec CNT100;
   1:  PR[91,1] = PR[90,1] + 2.723;
   1:  PR[91,2] = PR[90,2] + -2.436;
   1:  PR[91,3] = PR[90,3] + 7.998;
   1:L PR[91] R[100]mm/sec CNT100;
   1:  PR[91,1] = PR[90,1] + 2.837;
   1:  PR[91,2] = PR[90,2] + -2.832;
   1:  PR[91,3] = PR[90,3] + 8.000;
   1:L PR[91] R[100]mm/sec CNT100;
   1:  PR[91,1] = PR[90,1] + 3.008;
   1:  PR[91,2] = PR[90,2] + -3.593;
   1:  PR[91,3] = PR[90,3] + 8.003;
   1:L PR[91] R[100]mm/sec CNT100;
   1:  PR[91,1] = PR[90,1] + 3.230;
   1:  PR[91,2] = PR[90,2] + -4.399;
   1:  PR[91,3] = PR[90,3] + 8.008;
   1:L PR[91] R[100]mm/sec CNT100;
   1:  PR[91,1] = PR[90,1] + 3.493;
   1:  PR[91,2] = PR[90,2] + -5.192;
   1:  PR[91,3] = PR[90,3] + 8.013;
   1:L PR[91] R[100]mm/sec CNT100;
   1:  PR[91,1] = PR[90,1] + 3.796;
   1:  PR[91,2] = PR[90,2] + -5.974;
   1:  PR[91,3] = PR[90,3] + 8.018;
   1:L PR[91] R[100]mm/sec CNT100;
   1:  PR[91,1] = PR[90,1] + 4.138;
   1:  PR[91,2] = PR[90,2] + -6.743;
   1:  PR[91,3] = PR[90,3] + 8.023;
   1:L PR[91] R[100]mm/sec CNT100;
   1:  PR[91,1] = PR[90,1] + 4.519;
   1:  PR[91,2] = PR[90,2] + -7.496;
   1:  PR[91,3] = PR[90,3] + 8.028;
   1:L PR[91] R[100]mm/sec CNT100;
   1:  PR[91,1] = PR[90,1] + 4.937;
   1:  PR[91,2] = PR[90,2] + -8.231;
   1:  PR[91,3] = PR[90,3] + 8.033;
   1:L PR[91] R[100]mm/sec CNT100;
   1:  PR[91,1] = PR[90,1] + 5.397;
   1:  PR[91,2] = PR[90,2] + -8.953;
   1:  PR[91,3] = PR[90,3] + 8.039;
   1:L PR[91] R[100]mm/sec CNT100;
   1:  PR[91,1] = PR[90,1] + 5.873;
   1:  PR[91,2] = PR[90,2] + -9.626;
   1:  PR[91,3] = PR[90,3] + 8.044;
   1:L PR[91] R[100]mm/sec CNT100;
   1:  PR[91,1] = PR[90,1] + 6.382;
   1:  PR[91,2] = PR[90,2] + -10.276;
   1:  PR[91,3] = PR[90,3] + 8.049;
   1:L PR[91] R[100]mm/sec CNT100;
   1:  PR[91,1] = PR[90,1] + 7.001;
   1:  PR[91,2] = PR[90,2] + -10.987;
   1:  PR[91,3] = PR[90,3] + 8.054;
   1:L PR[91] R[100]mm/sec CNT100;
   1:  PR[91,1] = PR[90,1] + 7.494;
   1:  PR[91,2] = PR[90,2] + -11.501;
   1:  PR[91,3] = PR[90,3] + 8.060;
   1:L PR[91] R[100]mm/sec CNT100;
   1:  PR[91,1] = PR[90,1] + 8.093;
   1:  PR[91,2] = PR[90,2] + -12.071;
   1:  PR[91,3] = PR[90,3] + 8.064;
   1:L PR[91] R[100]mm/sec CNT100;
   1:  PR[91,1] = PR[90,1] + 8.720;
   1:  PR[91,2] = PR[90,2] + -12.612;
   1:  PR[91,3] = PR[90,3] + 8.069;
   1:L PR[91] R[100]mm/sec CNT100;
   1:  PR[91,1] = PR[90,1] + 9.372;
   1:  PR[91,2] = PR[90,2] + -13.121;
   1:  PR[91,3] = PR[90,3] + 8.074;
   1:L PR[91] R[100]mm/sec CNT100;
   1:  PR[91,1] = PR[90,1] + 10.049;
   1:  PR[91,2] = PR[90,2] + -13.599;
   1:  PR[91,3] = PR[90,3] + 8.079;
   1:L PR[91] R[100]mm/sec CNT100;
   1:  PR[91,1] = PR[90,1] + 10.748;
   1:  PR[91,2] = PR[90,2] + -14.044;
   1:  PR[91,3] = PR[90,3] + 8.084;
   1:L PR[91] R[100]mm/sec CNT100;
   1:  PR[91,1] = PR[90,1] + 11.470;
   1:  PR[91,2] = PR[90,2] + -14.455;
   1:  PR[91,3] = PR[90,3] + 8.089;
   1:L PR[91] R[100]mm/sec CNT100;
   1:  PR[91,1] = PR[90,1] + 12.210;
   1:  PR[91,2] = PR[90,2] + -14.830;
   1:  PR[91,3] = PR[90,3] + 8.094;
   1:L PR[91] R[100]mm/sec CNT100;
   1:  PR[91,1] = PR[90,1] + 12.968;
   1:  PR[91,2] = PR[90,2] + -15.170;
   1:  PR[91,3] = PR[90,3] + 8.099;
   1:L PR[91] R[100]mm/sec CNT100;
   1:  PR[91,1] = PR[90,1] + 13.743;
   1:  PR[91,2] = PR[90,2] + -15.474;
   1:  PR[91,3] = PR[90,3] + 8.104;
   1:L PR[91] R[100]mm/sec CNT100;
   1:  PR[91,1] = PR[90,1] + 14.532;
   1:  PR[91,2] = PR[90,2] + -15.739;
   1:  PR[91,3] = PR[90,3] + 8.110;
   1:L PR[91] R[100]mm/sec CNT100;
   1:  PR[91,1] = PR[90,1] + 15.333;
   1:  PR[91,2] = PR[90,2] + -15.967;
   1:  PR[91,3] = PR[90,3] + 8.115;
   1:L PR[91] R[100]mm/sec CNT100;
   1:  PR[91,1] = PR[90,1] + 16.145;
   1:  PR[91,2] = PR[90,2] + -16.155;
   1:  PR[91,3] = PR[90,3] + 8.120;
   1:L PR[91] R[100]mm/sec CNT100;
   1:  PR[91,1] = PR[90,1] + 16.966;
   1:  PR[91,2] = PR[90,2] + -16.304;
   1:  PR[91,3] = PR[90,3] + 8.125;
   1:L PR[91] R[100]mm/sec CNT100;
   1:  PR[91,1] = PR[90,1] + 17.793;
   1:  PR[91,2] = PR[90,2] + -16.414;
   1:  PR[91,3] = PR[90,3] + 8.130;
   1:L PR[91] R[100]mm/sec CNT100;
   1:  PR[91,1] = PR[90,1] + 18.626;
   1:  PR[91,2] = PR[90,2] + -16.483;
   1:  PR[91,3] = PR[90,3] + 8.135;
   1:L PR[91] R[100]mm/sec CNT100;
   1:  PR[91,1] = PR[90,1] + 19.466;
   1:  PR[91,2] = PR[90,2] + -16.511;
   1:  PR[91,3] = PR[90,3] + 8.140;
   1:L PR[91] R[100]mm/sec CNT100;
   1:  PR[91,1] = PR[90,1] + 20.308;
   1:  PR[91,2] = PR[90,2] + -16.499;
   1:  PR[91,3] = PR[90,3] + 8.145;
   1:L PR[91] R[100]mm/sec CNT100;
   1:  PR[91,1] = PR[90,1] + 21.149;
   1:  PR[91,2] = PR[90,2] + -16.445;
   1:  PR[91,3] = PR[90,3] + 8.150;
   1:L PR[91] R[100]mm/sec CNT100;
   1:  PR[91,1] = PR[90,1] + 21.985;
   1:  PR[91,2] = PR[90,2] + -16.349;
   1:  PR[91,3] = PR[90,3] + 8.156;
   1:L PR[91] R[100]mm/sec CNT100;
   1:  PR[91,1] = PR[90,1] + 22.816;
   1:  PR[91,2] = PR[90,2] + -16.213;
   1:  PR[91,3] = PR[90,3] + 8.161;
   1:L PR[91] R[100]mm/sec CNT100;
   1:  PR[91,1] = PR[90,1] + 23.638;
   1:  PR[91,2] = PR[90,2] + -16.036;
   1:  PR[91,3] = PR[90,3] + 8.166;
   1:L PR[91] R[100]mm/sec CNT100;
   1:  PR[91,1] = PR[90,1] + 24.451;
   1:  PR[91,2] = PR[90,2] + -15.819;
   1:  PR[91,3] = PR[90,3] + 8.171;
   1:L PR[91] R[100]mm/sec CNT100;
   1:  PR[91,1] = PR[90,1] + 25.252;
   1:  PR[91,2] = PR[90,2] + -15.563;
   1:  PR[91,3] = PR[90,3] + 8.176;
   1:L PR[91] R[100]mm/sec CNT100;
   1:  PR[91,1] = PR[90,1] + 26.039;
   1:  PR[91,2] = PR[90,2] + -15.267;
   1:  PR[91,3] = PR[90,3] + 8.181;
   1:L PR[91] R[100]mm/sec CNT100;
   1:  PR[91,1] = PR[90,1] + 26.810;
   1:  PR[91,2] = PR[90,2] + -14.933;
   1:  PR[91,3] = PR[90,3] + 8.186;
   1:L PR[91] R[100]mm/sec CNT100;
   1:  PR[91,1] = PR[90,1] + 27.564;
   1:  PR[91,2] = PR[90,2] + -14.562;
   1:  PR[91,3] = PR[90,3] + 8.192;
   1:L PR[91] R[100]mm/sec CNT100;
   1:  PR[91,1] = PR[90,1] + 28.298;
   1:  PR[91,2] = PR[90,2] + -14.154;
   1:  PR[91,3] = PR[90,3] + 8.197;
   1:L PR[91] R[100]mm/sec CNT100;
   1:  PR[91,1] = PR[90,1] + 29.011;
   1:  PR[91,2] = PR[90,2] + -13.711;
   1:  PR[91,3] = PR[90,3] + 8.202;
   1:L PR[91] R[100]mm/sec CNT100;
   1:  PR[91,1] = PR[90,1] + 29.701;
   1:  PR[91,2] = PR[90,2] + -13.233;
   1:  PR[91,3] = PR[90,3] + 8.207;
   1:L PR[91] R[100]mm/sec CNT100;
   1:  PR[91,1] = PR[90,1] + 30.366;
   1:  PR[91,2] = PR[90,2] + -12.722;
   1:  PR[91,3] = PR[90,3] + 8.212;
   1:L PR[91] R[100]mm/sec CNT100;
   1:  PR[91,1] = PR[90,1] + 31.005;
   1:  PR[91,2] = PR[90,2] + -12.179;
   1:  PR[91,3] = PR[90,3] + 8.217;
   1:L PR[91] R[100]mm/sec CNT100;
   1:  PR[91,1] = PR[90,1] + 31.617;
   1:  PR[91,2] = PR[90,2] + -11.606;
   1:  PR[91,3] = PR[90,3] + 8.222;
   1:L PR[91] R[100]mm/sec CNT100;
   1:  PR[91,1] = PR[90,1] + 32.199;
   1:  PR[91,2] = PR[90,2] + -11.002;
   1:  PR[91,3] = PR[90,3] + 8.227;
   1:L PR[91] R[100]mm/sec CNT100;
   1:  PR[91,1] = PR[90,1] + 32.750;
   1:  PR[91,2] = PR[90,2] + -10.370;
   1:  PR[91,3] = PR[90,3] + 8.233;
   1:L PR[91] R[100]mm/sec CNT100;
   1:  PR[91,1] = PR[90,1] + 33.269;
   1:  PR[91,2] = PR[90,2] + -9.713;
   1:  PR[91,3] = PR[90,3] + 8.238;
   1:L PR[91] R[100]mm/sec CNT100;
   1:  PR[91,1] = PR[90,1] + 33.756;
   1:  PR[91,2] = PR[90,2] + -9.030;
   1:  PR[91,3] = PR[90,3] + 8.243;
   1:L PR[91] R[100]mm/sec CNT100;
   1:  PR[91,1] = PR[90,1] + 34.207;
   1:  PR[91,2] = PR[90,2] + -8.324;
   1:  PR[91,3] = PR[90,3] + 8.248;
   1:L PR[91] R[100]mm/sec CNT100;
   1:  PR[91,1] = PR[90,1] + 34.624;
   1:  PR[91,2] = PR[90,2] + -7.597;
   1:  PR[91,3] = PR[90,3] + 8.253;
   1:L PR[91] R[100]mm/sec CNT100;
   1:  PR[91,1] = PR[90,1] + 35.003;
   1:  PR[91,2] = PR[90,2] + -6.851;
   1:  PR[91,3] = PR[90,3] + 8.258;
   1:L PR[91] R[100]mm/sec CNT100;
   1:  PR[91,1] = PR[90,1] + 35.345;
   1:  PR[91,2] = PR[90,2] + -6.088;
   1:  PR[91,3] = PR[90,3] + 8.263;
   1:L PR[91] R[100]mm/sec CNT100;
   1:  PR[91,1] = PR[90,1] + 35.649;
   1:  PR[91,2] = PR[90,2] + -5.310;
   1:  PR[91,3] = PR[90,3] + 8.268;
   1:L PR[91] R[100]mm/sec CNT100;
   1:  PR[91,1] = PR[90,1] + 35.914;
   1:  PR[91,2] = PR[90,2] + -4.519;
   1:  PR[91,3] = PR[90,3] + 8.274;
   1:L PR[91] R[100]mm/sec CNT100;
   1:  PR[91,1] = PR[90,1] + 36.139;
   1:  PR[91,2] = PR[90,2] + -3.716;
   1:  PR[91,3] = PR[90,3] + 8.279;
   1:L PR[91] R[100]mm/sec CNT100;
   1:  PR[91,1] = PR[90,1] + 36.324;
   1:  PR[91,2] = PR[90,2] + -2.903;
   1:  PR[91,3] = PR[90,3] + 8.284;
   1:L PR[91] R[100]mm/sec CNT100;
   1:  PR[91,1] = PR[90,1] + 36.469;
   1:  PR[91,2] = PR[90,2] + -2.081;
   1:  PR[91,3] = PR[90,3] + 8.289;
   1:L PR[91] R[100]mm/sec CNT100;
   1:  PR[91,1] = PR[90,1] + 36.572;
   1:  PR[91,2] = PR[90,2] + -1.251;
   1:  PR[91,3] = PR[90,3] + 8.294;
   1:L PR[91] R[100]mm/sec CNT100;
   1:  PR[91,1] = PR[90,1] + 36.634;
   1:  PR[91,2] = PR[90,2] + -0.414;
   1:  PR[91,3] = PR[90,3] + 8.299;
   1:L PR[91] R[100]mm/sec CNT100;
   1:  PR[91,1] = PR[90,1] + 36.656;
   1:  PR[91,2] = PR[90,2] + 0.428;
   1:  PR[91,3] = PR[90,3] + 8.304;
   1:L PR[91] R[100]mm/sec CNT100;
   1:  PR[91,1] = PR[90,1] + 36.634;
   1:  PR[91,2] = PR[90,2] + 1.269;
   1:  PR[91,3] = PR[90,3] + 8.309;
   1:L PR[91] R[100]mm/sec CNT100;
   1:  PR[91,1] = PR[90,1] + 36.572;
   1:  PR[91,2] = PR[90,2] + 2.106;
   1:  PR[91,3] = PR[90,3] + 8.314;
   1:L PR[91] R[100]mm/sec CNT100;
   1:  PR[91,1] = PR[90,1] + 36.469;
   1:  PR[91,2] = PR[90,2] + 2.936;
   1:  PR[91,3] = PR[90,3] + 8.320;
   1:L PR[91] R[100]mm/sec CNT100;
   1:  PR[91,1] = PR[90,1] + 36.324;
   1:  PR[91,2] = PR[90,2] + 3.759;
   1:  PR[91,3] = PR[90,3] + 8.325;
   1:L PR[91] R[100]mm/sec CNT100;
   1:  PR[91,1] = PR[90,1] + 36.139;
   1:  PR[91,2] = PR[90,2] + 4.571;
   1:  PR[91,3] = PR[90,3] + 8.330;
   1:L PR[91] R[100]mm/sec CNT100;
   1:  PR[91,1] = PR[90,1] + 35.914;
   1:  PR[91,2] = PR[90,2] + 5.374;
   1:  PR[91,3] = PR[90,3] + 8.335;
   1:L PR[91] R[100]mm/sec CNT100;
   1:  PR[91,1] = PR[90,1] + 35.649;
   1:  PR[91,2] = PR[90,2] + 6.165;
   1:  PR[91,3] = PR[90,3] + 8.340;
   1:L PR[91] R[100]mm/sec CNT100;
   1:  PR[91,1] = PR[90,1] + 35.346;
   1:  PR[91,2] = PR[90,2] + 6.943;
   1:  PR[91,3] = PR[90,3] + 8.345;
   1:L PR[91] R[100]mm/sec CNT100;
   1:  PR[91,1] = PR[90,1] + 35.003;
   1:  PR[91,2] = PR[90,2] + 7.706;
   1:  PR[91,3] = PR[90,3] + 8.350;
   1:L PR[91] R[100]mm/sec CNT100;
   1:  PR[91,1] = PR[90,1] + 34.623;
   1:  PR[91,2] = PR[90,2] + 8.452;
   1:  PR[91,3] = PR[90,3] + 8.355;
   1:L PR[91] R[100]mm/sec CNT100;
   1:  PR[91,1] = PR[90,1] + 34.207;
   1:  PR[91,2] = PR[90,2] + 9.179;
   1:  PR[91,3] = PR[90,3] + 8.360;
   1:L PR[91] R[100]mm/sec CNT100;
   1:  PR[91,1] = PR[90,1] + 33.756;
   1:  PR[91,2] = PR[90,2] + 9.885;
   1:  PR[91,3] = PR[90,3] + 8.366;
   1:L PR[91] R[100]mm/sec CNT100;
   1:  PR[91,1] = PR[90,1] + 33.269;
   1:  PR[91,2] = PR[90,2] + 10.568;
   1:  PR[91,3] = PR[90,3] + 8.371;
   1:L PR[91] R[100]mm/sec CNT100;
   1:  PR[91,1] = PR[90,1] + 32.750;
   1:  PR[91,2] = PR[90,2] + 11.226;
   1:  PR[91,3] = PR[90,3] + 8.376;
   1:L PR[91] R[100]mm/sec CNT100;
   1:  PR[91,1] = PR[90,1] + 32.199;
   1:  PR[91,2] = PR[90,2] + 11.857;
   1:  PR[91,3] = PR[90,3] + 8.381;
   1:L PR[91] R[100]mm/sec CNT100;
   1:  PR[91,1] = PR[90,1] + 31.617;
   1:  PR[91,2] = PR[90,2] + 12.461;
   1:  PR[91,3] = PR[90,3] + 8.386;
   1:L PR[91] R[100]mm/sec CNT100;
   1:  PR[91,1] = PR[90,1] + 31.005;
   1:  PR[91,2] = PR[90,2] + 13.035;
   1:  PR[91,3] = PR[90,3] + 8.391;
   1:L PR[91] R[100]mm/sec CNT100;
   1:  PR[91,1] = PR[90,1] + 30.366;
   1:  PR[91,2] = PR[90,2] + 13.578;
   1:  PR[91,3] = PR[90,3] + 8.396;
   1:L PR[91] R[100]mm/sec CNT100;
   1:  PR[91,1] = PR[90,1] + 29.701;
   1:  PR[91,2] = PR[90,2] + 14.089;
   1:  PR[91,3] = PR[90,3] + 8.401;
   1:L PR[91] R[100]mm/sec CNT100;
   1:  PR[91,1] = PR[90,1] + 29.011;
   1:  PR[91,2] = PR[90,2] + 14.566;
   1:  PR[91,3] = PR[90,3] + 8.406;
   1:L PR[91] R[100]mm/sec CNT100;
   1:  PR[91,1] = PR[90,1] + 28.298;
   1:  PR[91,2] = PR[90,2] + 15.009;
   1:  PR[91,3] = PR[90,3] + 8.412;
   1:L PR[91] R[100]mm/sec CNT100;
   1:  PR[91,1] = PR[90,1] + 27.564;
   1:  PR[91,2] = PR[90,2] + 15.417;
   1:  PR[91,3] = PR[90,3] + 8.417;
   1:L PR[91] R[100]mm/sec CNT100;
   1:  PR[91,1] = PR[90,1] + 26.810;
   1:  PR[91,2] = PR[90,2] + 15.788;
   1:  PR[91,3] = PR[90,3] + 8.422;
   1:L PR[91] R[100]mm/sec CNT100;
   1:  PR[91,1] = PR[90,1] + 26.039;
   1:  PR[91,2] = PR[90,2] + 16.122;
   1:  PR[91,3] = PR[90,3] + 8.427;
   1:L PR[91] R[100]mm/sec CNT100;
   1:  PR[91,1] = PR[90,1] + 25.252;
   1:  PR[91,2] = PR[90,2] + 16.418;
   1:  PR[91,3] = PR[90,3] + 8.432;
   1:L PR[91] R[100]mm/sec CNT100;
   1:  PR[91,1] = PR[90,1] + 24.451;
   1:  PR[91,2] = PR[90,2] + 16.674;
   1:  PR[91,3] = PR[90,3] + 8.437;
   1:L PR[91] R[100]mm/sec CNT100;
   1:  PR[91,1] = PR[90,1] + 23.638;
   1:  PR[91,2] = PR[90,2] + 16.892;
   1:  PR[91,3] = PR[90,3] + 8.442;
   1:L PR[91] R[100]mm/sec CNT100;
   1:  PR[91,1] = PR[90,1] + 22.816;
   1:  PR[91,2] = PR[90,2] + 17.068;
   1:  PR[91,3] = PR[90,3] + 8.448;
   1:L PR[91] R[100]mm/sec CNT100;
   1:  PR[91,1] = PR[90,1] + 21.985;
   1:  PR[91,2] = PR[90,2] + 17.205;
   1:  PR[91,3] = PR[90,3] + 8.453;
   1:L PR[91] R[100]mm/sec CNT100;
   1:  PR[91,1] = PR[90,1] + 21.149;
   1:  PR[91,2] = PR[90,2] + 17.300;
   1:  PR[91,3] = PR[90,3] + 8.458;
   1:L PR[91] R[100]mm/sec CNT100;
   1:  PR[91,1] = PR[90,1] + 20.308;
   1:  PR[91,2] = PR[90,2] + 17.354;
   1:  PR[91,3] = PR[90,3] + 8.463;
   1:L PR[91] R[100]mm/sec CNT100;
   1:  PR[91,1] = PR[90,1] + 19.466;
   1:  PR[91,2] = PR[90,2] + 17.366;
   1:  PR[91,3] = PR[90,3] + 8.468;
   1:L PR[91] R[100]mm/sec CNT100;
   1:  PR[91,1] = PR[90,1] + 18.615;
   1:  PR[91,2] = PR[90,2] + 17.337;
   1:  PR[91,3] = PR[90,3] + 8.473;
   1:L PR[91] R[100]mm/sec CNT100;
   1:  PR[91,1] = PR[90,1] + 17.793;
   1:  PR[91,2] = PR[90,2] + 17.269;
   1:  PR[91,3] = PR[90,3] + 8.479;
   1:L PR[91] R[100]mm/sec CNT100;
   1:  PR[91,1] = PR[90,1] + 16.966;
   1:  PR[91,2] = PR[90,2] + 17.160;
   1:  PR[91,3] = PR[90,3] + 8.484;
   1:L PR[91] R[100]mm/sec CNT100;
   1:  PR[91,1] = PR[90,1] + 16.145;
   1:  PR[91,2] = PR[90,2] + 17.011;
   1:  PR[91,3] = PR[90,3] + 8.489;
   1:L PR[91] R[100]mm/sec CNT100;
   1:  PR[91,1] = PR[90,1] + 15.333;
   1:  PR[91,2] = PR[90,2] + 16.822;
   1:  PR[91,3] = PR[90,3] + 8.494;
   1:L PR[91] R[100]mm/sec CNT100;
   1:  PR[91,1] = PR[90,1] + 14.535;
   1:  PR[91,2] = PR[90,2] + 16.595;
   1:  PR[91,3] = PR[90,3] + 8.499;
   1:L PR[91] R[100]mm/sec CNT100;
   1:  PR[91,1] = PR[90,1] + 13.465;
   1:  PR[91,2] = PR[90,2] + 16.222;
   1:  PR[91,3] = PR[90,3] + 8.504;
   1:L PR[91] R[100]mm/sec CNT100;
   1:  PR[91,1] = PR[90,1] + 12.970;
   1:  PR[91,2] = PR[90,2] + 16.026;
   1:  PR[91,3] = PR[90,3] + 8.511;
   1:L PR[91] R[100]mm/sec CNT100;
   1:  PR[91,1] = PR[90,1] + 12.210;
   1:  PR[91,2] = PR[90,2] + 15.686;
   1:  PR[91,3] = PR[90,3] + 8.514;
   1:L PR[91] R[100]mm/sec CNT100;
   1:  PR[91,1] = PR[90,1] + 11.469;
   1:  PR[91,2] = PR[90,2] + 15.310;
   1:  PR[91,3] = PR[90,3] + 8.519;
   1:L PR[91] R[100]mm/sec CNT100;
   1:  PR[91,1] = PR[90,1] + 10.749;
   1:  PR[91,2] = PR[90,2] + 14.899;
   1:  PR[91,3] = PR[90,3] + 8.524;
   1:L PR[91] R[100]mm/sec CNT100;
   1:  PR[91,1] = PR[90,1] + 10.049;
   1:  PR[91,2] = PR[90,2] + 14.454;
   1:  PR[91,3] = PR[90,3] + 8.529;
   1:L PR[91] R[100]mm/sec CNT100;
   1:  PR[91,1] = PR[90,1] + 9.372;
   1:  PR[91,2] = PR[90,2] + 13.977;
   1:  PR[91,3] = PR[90,3] + 8.534;
   1:L PR[91] R[100]mm/sec CNT100;
   1:  PR[91,1] = PR[90,1] + 8.720;
   1:  PR[91,2] = PR[90,2] + 13.467;
   1:  PR[91,3] = PR[90,3] + 8.539;
   1:L PR[91] R[100]mm/sec CNT100;
   1:  PR[91,1] = PR[90,1] + 8.093;
   1:  PR[91,2] = PR[90,2] + 12.926;
   1:  PR[91,3] = PR[90,3] + 8.545;
   1:L PR[91] R[100]mm/sec CNT100;
   1:  PR[91,1] = PR[90,1] + 7.608;
   1:  PR[91,2] = PR[90,2] + 12.468;
   1:  PR[91,3] = PR[90,3] + 8.550;
   1:L PR[91] R[100]mm/sec CNT100;
   1:  PR[91,1] = PR[90,1] + 6.922;
   1:  PR[91,2] = PR[90,2] + 11.757;
   1:  PR[91,3] = PR[90,3] + 8.554;
   1:L PR[91] R[100]mm/sec CNT100;
   1:  PR[91,1] = PR[90,1] + 6.382;
   1:  PR[91,2] = PR[90,2] + 11.133;
   1:  PR[91,3] = PR[90,3] + 8.560;
   1:L PR[91] R[100]mm/sec CNT100;
   1:  PR[91,1] = PR[90,1] + 5.873;
   1:  PR[91,2] = PR[90,2] + 10.481;
   1:  PR[91,3] = PR[90,3] + 8.565;
   1:L PR[91] R[100]mm/sec CNT100;
   1:  PR[91,1] = PR[90,1] + 5.392;
   1:  PR[91,2] = PR[90,2] + 9.801;
   1:  PR[91,3] = PR[90,3] + 8.570;
   1:L PR[91] R[100]mm/sec CNT100;
   1:  PR[91,1] = PR[90,1] + 4.937;
   1:  PR[91,2] = PR[90,2] + 9.086;
   1:  PR[91,3] = PR[90,3] + 8.575;
   1:L PR[91] R[100]mm/sec CNT100;
   1:  PR[91,1] = PR[90,1] + 4.519;
   1:  PR[91,2] = PR[90,2] + 8.351;
   1:  PR[91,3] = PR[90,3] + 8.580;
   1:L PR[91] R[100]mm/sec CNT100;
   1:  PR[91,1] = PR[90,1] + 4.138;
   1:  PR[91,2] = PR[90,2] + 7.598;
   1:  PR[91,3] = PR[90,3] + 8.585;
   1:L PR[91] R[100]mm/sec CNT100;
   1:  PR[91,1] = PR[90,1] + 3.850;
   1:  PR[91,2] = PR[90,2] + 6.955;
   1:  PR[91,3] = PR[90,3] + 8.590;
   1:L PR[91] R[100]mm/sec CNT100;
   1:  PR[91,1] = PR[90,1] + 3.492;
   1:  PR[91,2] = PR[90,2] + 6.046;
   1:  PR[91,3] = PR[90,3] + 8.595;
   1:L PR[91] R[100]mm/sec CNT100;
   1:  PR[91,1] = PR[90,1] + 3.230;
   1:  PR[91,2] = PR[90,2] + 5.254;
   1:  PR[91,3] = PR[90,3] + 8.601;
   1:L PR[91] R[100]mm/sec CNT100;
   1:  PR[91,1] = PR[90,1] + 3.008;
   1:  PR[91,2] = PR[90,2] + 4.448;
   1:  PR[91,3] = PR[90,3] + 8.606;
   1:L PR[91] R[100]mm/sec CNT100;
   1:  PR[91,1] = PR[90,1] + 2.834;
   1:  PR[91,2] = PR[90,2] + 3.674;
   1:  PR[91,3] = PR[90,3] + 8.611;
   1:L PR[91] R[100]mm/sec CNT100;
   1:  PR[91,1] = PR[90,1] + 2.720;
   1:  PR[91,2] = PR[90,2] + 3.281;
   1:  PR[91,3] = PR[90,3] + 8.616;
   1:L PR[91] R[100]mm/sec CNT100;
   1:  PR[91,1] = PR[90,1] + 2.585;
   1:  PR[91,2] = PR[90,2] + 2.934;
   1:  PR[91,3] = PR[90,3] + 8.618;
   1:L PR[91] R[100]mm/sec CNT100;
   1:  PR[91,1] = PR[90,1] + 2.354;
   1:  PR[91,2] = PR[90,2] + 2.483;
   1:  PR[91,3] = PR[90,3] + 8.620;
   1:L PR[91] R[100]mm/sec CNT100;
   1:  PR[91,1] = PR[90,1] + 2.086;
   1:  PR[91,2] = PR[90,2] + 2.110;
   1:  PR[91,3] = PR[90,3] + 8.624;
   1:L PR[91] R[100]mm/sec CNT100;
   1:  PR[91,1] = PR[90,1] + 1.894;
   1:  PR[91,2] = PR[90,2] + 1.899;
   1:  PR[91,3] = PR[90,3] + 8.626;
   1:L PR[91] R[100]mm/sec CNT100;
   1:  PR[91,1] = PR[90,1] + 1.669;
   1:  PR[91,2] = PR[90,2] + 1.693;
   1:  PR[91,3] = PR[90,3] + 8.628;
   1:L PR[91] R[100]mm/sec CNT100;
   1:  PR[91,1] = PR[90,1] + 1.393;
   1:  PR[91,2] = PR[90,2] + 1.497;
   1:  PR[91,3] = PR[90,3] + 8.630;
   1:L PR[91] R[100]mm/sec CNT100;
   1:  PR[91,1] = PR[90,1] + 1.087;
   1:  PR[91,2] = PR[90,2] + 1.340;
   1:  PR[91,3] = PR[90,3] + 8.632;
   1:L PR[91] R[100]mm/sec CNT100;
   1:  PR[91,1] = PR[90,1] + 0.673;
   1:  PR[91,2] = PR[90,2] + 1.169;
   1:  PR[91,3] = PR[90,3] + 8.634;
   1:L PR[91] R[100]mm/sec CNT100;
   1:  PR[91,1] = PR[90,1] + -0.010;
   1:  PR[91,2] = PR[90,2] + 1.064;
   1:  PR[91,3] = PR[90,3] + 8.637;
   1:L PR[91] R[100]mm/sec CNT100;
   1:  PR[91,1] = PR[90,1] + -0.643;
   1:  PR[91,2] = PR[90,2] + 1.113;
   1:  PR[91,3] = PR[90,3] + 8.641;
   1:L PR[91] R[100]mm/sec CNT100;
   1:  PR[91,1] = PR[90,1] + -1.215;
   1:  PR[91,2] = PR[90,2] + 1.283;
   1:  PR[91,3] = PR[90,3] + 8.645;
   1:L PR[91] R[100]mm/sec CNT100;
   1:  PR[91,1] = PR[90,1] + -1.380;
   1:  PR[91,2] = PR[90,2] + 1.365;
   1:  PR[91,3] = PR[90,3] + 8.649;
   1:L PR[91] R[100]mm/sec CNT100;
   1:  PR[91,1] = PR[90,1] + -1.748;
   1:  PR[91,2] = PR[90,2] + 1.574;
   1:  PR[91,3] = PR[90,3] + 8.650;
   1:L PR[91] R[100]mm/sec CNT100;
   1:  PR[91,1] = PR[90,1] + -2.196;
   1:  PR[91,2] = PR[90,2] + 1.950;
   1:  PR[91,3] = PR[90,3] + 8.652;
   1:L PR[91] R[100]mm/sec CNT100;
   1:  PR[91,1] = PR[90,1] + -2.536;
   1:  PR[91,2] = PR[90,2] + 2.392;
   1:  PR[91,3] = PR[90,3] + 8.656;
   1:L PR[91] R[100]mm/sec CNT100;
   1:  PR[91,1] = PR[90,1] + -2.690;
   1:  PR[91,2] = PR[90,2] + 2.654;
   1:  PR[91,3] = PR[90,3] + 8.659;
   1:L PR[91] R[100]mm/sec CNT100;
   1:  PR[91,1] = PR[90,1] + -2.827;
   1:  PR[91,2] = PR[90,2] + 2.939;
   1:  PR[91,3] = PR[90,3] + 8.661;
   1:L PR[91] R[100]mm/sec CNT100;
   1:  PR[91,1] = PR[90,1] + -2.962;
   1:  PR[91,2] = PR[90,2] + 3.290;
   1:  PR[91,3] = PR[90,3] + 8.663;
   1:L PR[91] R[100]mm/sec CNT100;
   1:  PR[91,1] = PR[90,1] + -3.076;
   1:  PR[91,2] = PR[90,2] + 3.686;
   1:  PR[91,3] = PR[90,3] + 8.665;
   1:L PR[91] R[100]mm/sec CNT100;
   1:  PR[91,1] = PR[90,1] + -3.247;
   1:  PR[91,2] = PR[90,2] + 4.447;
   1:  PR[91,3] = PR[90,3] + 8.668;
   1:L PR[91] R[100]mm/sec CNT100;
   1:  PR[91,1] = PR[90,1] + -3.470;
   1:  PR[91,2] = PR[90,2] + 5.253;
   1:  PR[91,3] = PR[90,3] + 8.673;
   1:L PR[91] R[100]mm/sec CNT100;
   1:  PR[91,1] = PR[90,1] + -3.733;
   1:  PR[91,2] = PR[90,2] + 6.048;
   1:  PR[91,3] = PR[90,3] + 8.678;
   1:L PR[91] R[100]mm/sec CNT100;
   1:  PR[91,1] = PR[90,1] + -4.036;
   1:  PR[91,2] = PR[90,2] + 6.831;
   1:  PR[91,3] = PR[90,3] + 8.683;
   1:L PR[91] R[100]mm/sec CNT100;
   1:  PR[91,1] = PR[90,1] + -4.378;
   1:  PR[91,2] = PR[90,2] + 7.602;
   1:  PR[91,3] = PR[90,3] + 8.688;
   1:L PR[91] R[100]mm/sec CNT100;
   1:  PR[91,1] = PR[90,1] + -4.759;
   1:  PR[91,2] = PR[90,2] + 8.356;
   1:  PR[91,3] = PR[90,3] + 8.693;
   1:L PR[91] R[100]mm/sec CNT100;
   1:  PR[91,1] = PR[90,1] + -5.177;
   1:  PR[91,2] = PR[90,2] + 9.091;
   1:  PR[91,3] = PR[90,3] + 8.698;
   1:L PR[91] R[100]mm/sec CNT100;
   1:  PR[91,1] = PR[90,1] + -5.637;
   1:  PR[91,2] = PR[90,2] + 9.813;
   1:  PR[91,3] = PR[90,3] + 8.704;
   1:L PR[91] R[100]mm/sec CNT100;
   1:  PR[91,1] = PR[90,1] + -6.113;
   1:  PR[91,2] = PR[90,2] + 10.485;
   1:  PR[91,3] = PR[90,3] + 8.709;
   1:L PR[91] R[100]mm/sec CNT100;
   1:  PR[91,1] = PR[90,1] + -6.622;
   1:  PR[91,2] = PR[90,2] + 11.136;
   1:  PR[91,3] = PR[90,3] + 8.714;
   1:L PR[91] R[100]mm/sec CNT100;
   1:  PR[91,1] = PR[90,1] + -7.163;
   1:  PR[91,2] = PR[90,2] + 11.761;
   1:  PR[91,3] = PR[90,3] + 8.719;
   1:L PR[91] R[100]mm/sec CNT100;
   1:  PR[91,1] = PR[90,1] + -7.734;
   1:  PR[91,2] = PR[90,2] + 12.358;
   1:  PR[91,3] = PR[90,3] + 8.724;
   1:L PR[91] R[100]mm/sec CNT100;
   1:  PR[91,1] = PR[90,1] + -8.333;
   1:  PR[91,2] = PR[90,2] + 12.928;
   1:  PR[91,3] = PR[90,3] + 8.729;
   1:L PR[91] R[100]mm/sec CNT100;
   1:  PR[91,1] = PR[90,1] + -8.960;
   1:  PR[91,2] = PR[90,2] + 13.468;
   1:  PR[91,3] = PR[90,3] + 8.734;
   1:L PR[91] R[100]mm/sec CNT100;
   1:  PR[91,1] = PR[90,1] + -9.612;
   1:  PR[91,2] = PR[90,2] + 13.977;
   1:  PR[91,3] = PR[90,3] + 8.739;
   1:L PR[91] R[100]mm/sec CNT100;
   1:  PR[91,1] = PR[90,1] + -10.289;
   1:  PR[91,2] = PR[90,2] + 14.455;
   1:  PR[91,3] = PR[90,3] + 8.744;
   1:L PR[91] R[100]mm/sec CNT100;
   1:  PR[91,1] = PR[90,1] + -10.989;
   1:  PR[91,2] = PR[90,2] + 14.900;
   1:  PR[91,3] = PR[90,3] + 8.749;
   1:L PR[91] R[100]mm/sec CNT100;
   1:  PR[91,1] = PR[90,1] + -11.710;
   1:  PR[91,2] = PR[90,2] + 15.310;
   1:  PR[91,3] = PR[90,3] + 8.754;
   1:L PR[91] R[100]mm/sec CNT100;
   1:  PR[91,1] = PR[90,1] + -12.450;
   1:  PR[91,2] = PR[90,2] + 15.686;
   1:  PR[91,3] = PR[90,3] + 8.759;
   1:L PR[91] R[100]mm/sec CNT100;
   1:  PR[91,1] = PR[90,1] + -13.208;
   1:  PR[91,2] = PR[90,2] + 16.026;
   1:  PR[91,3] = PR[90,3] + 8.764;
   1:L PR[91] R[100]mm/sec CNT100;
   1:  PR[91,1] = PR[90,1] + -13.983;
   1:  PR[91,2] = PR[90,2] + 16.330;
   1:  PR[91,3] = PR[90,3] + 8.769;
   1:L PR[91] R[100]mm/sec CNT100;
   1:  PR[91,1] = PR[90,1] + -14.771;
   1:  PR[91,2] = PR[90,2] + 16.595;
   1:  PR[91,3] = PR[90,3] + 8.775;
   1:L PR[91] R[100]mm/sec CNT100;
   1:  PR[91,1] = PR[90,1] + -15.573;
   1:  PR[91,2] = PR[90,2] + 16.823;
   1:  PR[91,3] = PR[90,3] + 8.780;
   1:L PR[91] R[100]mm/sec CNT100;
   1:  PR[91,1] = PR[90,1] + -16.385;
   1:  PR[91,2] = PR[90,2] + 17.011;
   1:  PR[91,3] = PR[90,3] + 8.785;
   1:L PR[91] R[100]mm/sec CNT100;
   1:  PR[91,1] = PR[90,1] + -17.205;
   1:  PR[91,2] = PR[90,2] + 17.160;
   1:  PR[91,3] = PR[90,3] + 8.790;
   1:L PR[91] R[100]mm/sec CNT100;
   1:  PR[91,1] = PR[90,1] + -18.033;
   1:  PR[91,2] = PR[90,2] + 17.269;
   1:  PR[91,3] = PR[90,3] + 8.795;
   1:L PR[91] R[100]mm/sec CNT100;
   1:  PR[91,1] = PR[90,1] + -18.865;
   1:  PR[91,2] = PR[90,2] + 17.338;
   1:  PR[91,3] = PR[90,3] + 8.800;
   1:L PR[91] R[100]mm/sec CNT100;
   1:  PR[91,1] = PR[90,1] + -19.705;
   1:  PR[91,2] = PR[90,2] + 17.366;
   1:  PR[91,3] = PR[90,3] + 8.805;
   1:L PR[91] R[100]mm/sec CNT100;
   1:  PR[91,1] = PR[90,1] + -20.547;
   1:  PR[91,2] = PR[90,2] + 17.354;
   1:  PR[91,3] = PR[90,3] + 8.810;
   1:L PR[91] R[100]mm/sec CNT100;
   1:  PR[91,1] = PR[90,1] + -21.388;
   1:  PR[91,2] = PR[90,2] + 17.300;
   1:  PR[91,3] = PR[90,3] + 8.815;
   1:L PR[91] R[100]mm/sec CNT100;
   1:  PR[91,1] = PR[90,1] + -22.224;
   1:  PR[91,2] = PR[90,2] + 17.204;
   1:  PR[91,3] = PR[90,3] + 8.821;
   1:L PR[91] R[100]mm/sec CNT100;
   1:  PR[91,1] = PR[90,1] + -23.055;
   1:  PR[91,2] = PR[90,2] + 17.068;
   1:  PR[91,3] = PR[90,3] + 8.826;
   1:L PR[91] R[100]mm/sec CNT100;
   1:  PR[91,1] = PR[90,1] + -23.878;
   1:  PR[91,2] = PR[90,2] + 16.892;
   1:  PR[91,3] = PR[90,3] + 8.831;
   1:L PR[91] R[100]mm/sec CNT100;
   1:  PR[91,1] = PR[90,1] + -24.690;
   1:  PR[91,2] = PR[90,2] + 16.675;
   1:  PR[91,3] = PR[90,3] + 8.836;
   1:L PR[91] R[100]mm/sec CNT100;
   1:  PR[91,1] = PR[90,1] + -25.491;
   1:  PR[91,2] = PR[90,2] + 16.418;
   1:  PR[91,3] = PR[90,3] + 8.841;
   1:L PR[91] R[100]mm/sec CNT100;
   1:  PR[91,1] = PR[90,1] + -26.278;
   1:  PR[91,2] = PR[90,2] + 16.122;
   1:  PR[91,3] = PR[90,3] + 8.846;
   1:L PR[91] R[100]mm/sec CNT100;
   1:  PR[91,1] = PR[90,1] + -27.049;
   1:  PR[91,2] = PR[90,2] + 15.788;
   1:  PR[91,3] = PR[90,3] + 8.851;
   1:L PR[91] R[100]mm/sec CNT100;
   1:  PR[91,1] = PR[90,1] + -27.803;
   1:  PR[91,2] = PR[90,2] + 15.417;
   1:  PR[91,3] = PR[90,3] + 8.857;
   1:L PR[91] R[100]mm/sec CNT100;
   1:  PR[91,1] = PR[90,1] + -28.537;
   1:  PR[91,2] = PR[90,2] + 15.009;
   1:  PR[91,3] = PR[90,3] + 8.862;
   1:L PR[91] R[100]mm/sec CNT100;
   1:  PR[91,1] = PR[90,1] + -29.250;
   1:  PR[91,2] = PR[90,2] + 14.566;
   1:  PR[91,3] = PR[90,3] + 8.867;
   1:L PR[91] R[100]mm/sec CNT100;
   1:  PR[91,1] = PR[90,1] + -29.940;
   1:  PR[91,2] = PR[90,2] + 14.088;
   1:  PR[91,3] = PR[90,3] + 8.872;
   1:L PR[91] R[100]mm/sec CNT100;
   1:  PR[91,1] = PR[90,1] + -30.605;
   1:  PR[91,2] = PR[90,2] + 13.577;
   1:  PR[91,3] = PR[90,3] + 8.877;
   1:L PR[91] R[100]mm/sec CNT100;
   1:  PR[91,1] = PR[90,1] + -31.244;
   1:  PR[91,2] = PR[90,2] + 13.034;
   1:  PR[91,3] = PR[90,3] + 8.882;
   1:L PR[91] R[100]mm/sec CNT100;
   1:  PR[91,1] = PR[90,1] + -31.855;
   1:  PR[91,2] = PR[90,2] + 12.460;
   1:  PR[91,3] = PR[90,3] + 8.887;
   1:L PR[91] R[100]mm/sec CNT100;
   1:  PR[91,1] = PR[90,1] + -32.438;
   1:  PR[91,2] = PR[90,2] + 11.857;
   1:  PR[91,3] = PR[90,3] + 8.892;
   1:L PR[91] R[100]mm/sec CNT100;
   1:  PR[91,1] = PR[90,1] + -32.989;
   1:  PR[91,2] = PR[90,2] + 11.226;
   1:  PR[91,3] = PR[90,3] + 8.898;
   1:L PR[91] R[100]mm/sec CNT100;
   1:  PR[91,1] = PR[90,1] + -33.508;
   1:  PR[91,2] = PR[90,2] + 10.568;
   1:  PR[91,3] = PR[90,3] + 8.903;
   1:L PR[91] R[100]mm/sec CNT100;
   1:  PR[91,1] = PR[90,1] + -33.994;
   1:  PR[91,2] = PR[90,2] + 9.886;
   1:  PR[91,3] = PR[90,3] + 8.908;
   1:L PR[91] R[100]mm/sec CNT100;
   1:  PR[91,1] = PR[90,1] + -34.446;
   1:  PR[91,2] = PR[90,2] + 9.180;
   1:  PR[91,3] = PR[90,3] + 8.913;
   1:L PR[91] R[100]mm/sec CNT100;
   1:  PR[91,1] = PR[90,1] + -34.862;
   1:  PR[91,2] = PR[90,2] + 8.453;
   1:  PR[91,3] = PR[90,3] + 8.918;
   1:L PR[91] R[100]mm/sec CNT100;
   1:  PR[91,1] = PR[90,1] + -35.242;
   1:  PR[91,2] = PR[90,2] + 7.706;
   1:  PR[91,3] = PR[90,3] + 8.923;
   1:L PR[91] R[100]mm/sec CNT100;
   1:  PR[91,1] = PR[90,1] + -35.584;
   1:  PR[91,2] = PR[90,2] + 6.942;
   1:  PR[91,3] = PR[90,3] + 8.928;
   1:L PR[91] R[100]mm/sec CNT100;
   1:  PR[91,1] = PR[90,1] + -35.888;
   1:  PR[91,2] = PR[90,2] + 6.164;
   1:  PR[91,3] = PR[90,3] + 8.933;
   1:L PR[91] R[100]mm/sec CNT100;
   1:  PR[91,1] = PR[90,1] + -36.153;
   1:  PR[91,2] = PR[90,2] + 5.372;
   1:  PR[91,3] = PR[90,3] + 8.939;
   1:L PR[91] R[100]mm/sec CNT100;
   1:  PR[91,1] = PR[90,1] + -36.378;
   1:  PR[91,2] = PR[90,2] + 4.570;
   1:  PR[91,3] = PR[90,3] + 8.944;
   1:L PR[91] R[100]mm/sec CNT100;
   1:  PR[91,1] = PR[90,1] + -36.563;
   1:  PR[91,2] = PR[90,2] + 3.757;
   1:  PR[91,3] = PR[90,3] + 8.949;
   1:L PR[91] R[100]mm/sec CNT100;
   1:  PR[91,1] = PR[90,1] + -36.707;
   1:  PR[91,2] = PR[90,2] + 2.935;
   1:  PR[91,3] = PR[90,3] + 8.954;
   1:L PR[91] R[100]mm/sec CNT100;
   1:  PR[91,1] = PR[90,1] + -36.811;
   1:  PR[91,2] = PR[90,2] + 2.106;
   1:  PR[91,3] = PR[90,3] + 8.959;
   1:L PR[91] R[100]mm/sec CNT100;
   1:  PR[91,1] = PR[90,1] + -36.873;
   1:  PR[91,2] = PR[90,2] + 1.269;
   1:  PR[91,3] = PR[90,3] + 8.964;
   1:L PR[91] R[100]mm/sec CNT100;
   1:  PR[91,1] = PR[90,1] + -36.895;
   1:  PR[91,2] = PR[90,2] + 0.428;
   1:  PR[91,3] = PR[90,3] + 8.969;
   1:L PR[91] R[100]mm/sec CNT100;
   1:  PR[91,1] = PR[90,1] + -36.873;
   1:  PR[91,2] = PR[90,2] + -0.414;
   1:  PR[91,3] = PR[90,3] + 8.974;
   1:L PR[91] R[100]mm/sec CNT100;
   1:  PR[91,1] = PR[90,1] + -36.811;
   1:  PR[91,2] = PR[90,2] + -1.251;
   1:  PR[91,3] = PR[90,3] + 8.979;
   1:L PR[91] R[100]mm/sec CNT100;
   1:  PR[91,1] = PR[90,1] + -36.707;
   1:  PR[91,2] = PR[90,2] + -2.080;
   1:  PR[91,3] = PR[90,3] + 8.985;
   1:L PR[91] R[100]mm/sec CNT100;
   1:  PR[91,1] = PR[90,1] + -36.563;
   1:  PR[91,2] = PR[90,2] + -2.901;
   1:  PR[91,3] = PR[90,3] + 8.990;
   1:L PR[91] R[100]mm/sec CNT100;
   1:  PR[91,1] = PR[90,1] + -36.378;
   1:  PR[91,2] = PR[90,2] + -3.714;
   1:  PR[91,3] = PR[90,3] + 8.995;
   1:L PR[91] R[100]mm/sec CNT100;
   1:  PR[91,1] = PR[90,1] + -36.153;
   1:  PR[91,2] = PR[90,2] + -4.517;
   1:  PR[91,3] = PR[90,3] + 9.000;
   1:L PR[91] R[100]mm/sec CNT100;
   1:  PR[91,1] = PR[90,1] + -35.888;
   1:  PR[91,2] = PR[90,2] + -5.309;
   1:  PR[91,3] = PR[90,3] + 9.005;
   1:L PR[91] R[100]mm/sec CNT100;
   1:  PR[91,1] = PR[90,1] + -35.584;
   1:  PR[91,2] = PR[90,2] + -6.087;
   1:  PR[91,3] = PR[90,3] + 9.010;
   1:L PR[91] R[100]mm/sec CNT100;
   1:  PR[91,1] = PR[90,1] + -35.242;
   1:  PR[91,2] = PR[90,2] + -6.851;
   1:  PR[91,3] = PR[90,3] + 9.015;
   1:L PR[91] R[100]mm/sec CNT100;
   1:  PR[91,1] = PR[90,1] + -34.862;
   1:  PR[91,2] = PR[90,2] + -7.597;
   1:  PR[91,3] = PR[90,3] + 9.020;
   1:L PR[91] R[100]mm/sec CNT100;
   1:  PR[91,1] = PR[90,1] + -34.446;
   1:  PR[91,2] = PR[90,2] + -8.325;
   1:  PR[91,3] = PR[90,3] + 9.025;
   1:L PR[91] R[100]mm/sec CNT100;
   1:  PR[91,1] = PR[90,1] + -33.994;
   1:  PR[91,2] = PR[90,2] + -9.031;
   1:  PR[91,3] = PR[90,3] + 9.031;
   1:L PR[91] R[100]mm/sec CNT100;
   1:  PR[91,1] = PR[90,1] + -33.508;
   1:  PR[91,2] = PR[90,2] + -9.713;
   1:  PR[91,3] = PR[90,3] + 9.036;
   1:L PR[91] R[100]mm/sec CNT100;
   1:  PR[91,1] = PR[90,1] + -32.989;
   1:  PR[91,2] = PR[90,2] + -10.371;
   1:  PR[91,3] = PR[90,3] + 9.041;
   1:L PR[91] R[100]mm/sec CNT100;
   1:  PR[91,1] = PR[90,1] + -32.438;
   1:  PR[91,2] = PR[90,2] + -11.002;
   1:  PR[91,3] = PR[90,3] + 9.046;
   1:L PR[91] R[100]mm/sec CNT100;
   1:  PR[91,1] = PR[90,1] + -31.855;
   1:  PR[91,2] = PR[90,2] + -11.605;
   1:  PR[91,3] = PR[90,3] + 9.051;
   1:L PR[91] R[100]mm/sec CNT100;
   1:  PR[91,1] = PR[90,1] + -31.244;
   1:  PR[91,2] = PR[90,2] + -12.179;
   1:  PR[91,3] = PR[90,3] + 9.056;
   1:L PR[91] R[100]mm/sec CNT100;
   1:  PR[91,1] = PR[90,1] + -30.605;
   1:  PR[91,2] = PR[90,2] + -12.722;
   1:  PR[91,3] = PR[90,3] + 9.061;
   1:L PR[91] R[100]mm/sec CNT100;
   1:  PR[91,1] = PR[90,1] + -29.940;
   1:  PR[91,2] = PR[90,2] + -13.233;
   1:  PR[91,3] = PR[90,3] + 9.066;
   1:L PR[91] R[100]mm/sec CNT100;
   1:  PR[91,1] = PR[90,1] + -29.250;
   1:  PR[91,2] = PR[90,2] + -13.710;
   1:  PR[91,3] = PR[90,3] + 9.071;
   1:L PR[91] R[100]mm/sec CNT100;
   1:  PR[91,1] = PR[90,1] + -28.537;
   1:  PR[91,2] = PR[90,2] + -14.154;
   1:  PR[91,3] = PR[90,3] + 9.077;
   1:L PR[91] R[100]mm/sec CNT100;
   1:  PR[91,1] = PR[90,1] + -27.803;
   1:  PR[91,2] = PR[90,2] + -14.562;
   1:  PR[91,3] = PR[90,3] + 9.082;
   1:L PR[91] R[100]mm/sec CNT100;
   1:  PR[91,1] = PR[90,1] + -27.049;
   1:  PR[91,2] = PR[90,2] + -14.933;
   1:  PR[91,3] = PR[90,3] + 9.087;
   1:L PR[91] R[100]mm/sec CNT100;
   1:  PR[91,1] = PR[90,1] + -26.278;
   1:  PR[91,2] = PR[90,2] + -15.267;
   1:  PR[91,3] = PR[90,3] + 9.092;
   1:L PR[91] R[100]mm/sec CNT100;
   1:  PR[91,1] = PR[90,1] + -25.491;
   1:  PR[91,2] = PR[90,2] + -15.563;
   1:  PR[91,3] = PR[90,3] + 9.097;
   1:L PR[91] R[100]mm/sec CNT100;
   1:  PR[91,1] = PR[90,1] + -24.690;
   1:  PR[91,2] = PR[90,2] + -15.819;
   1:  PR[91,3] = PR[90,3] + 9.102;
   1:L PR[91] R[100]mm/sec CNT100;
   1:  PR[91,1] = PR[90,1] + -23.878;
   1:  PR[91,2] = PR[90,2] + -16.036;
   1:  PR[91,3] = PR[90,3] + 9.107;
   1:L PR[91] R[100]mm/sec CNT100;
   1:  PR[91,1] = PR[90,1] + -23.055;
   1:  PR[91,2] = PR[90,2] + -16.213;
   1:  PR[91,3] = PR[90,3] + 9.113;
   1:L PR[91] R[100]mm/sec CNT100;
   1:  PR[91,1] = PR[90,1] + -22.224;
   1:  PR[91,2] = PR[90,2] + -16.349;
   1:  PR[91,3] = PR[90,3] + 9.118;
   1:L PR[91] R[100]mm/sec CNT100;
   1:  PR[91,1] = PR[90,1] + -21.388;
   1:  PR[91,2] = PR[90,2] + -16.444;
   1:  PR[91,3] = PR[90,3] + 9.123;
   1:L PR[91] R[100]mm/sec CNT100;
   1:  PR[91,1] = PR[90,1] + -20.547;
   1:  PR[91,2] = PR[90,2] + -16.498;
   1:  PR[91,3] = PR[90,3] + 9.128;
   1:L PR[91] R[100]mm/sec CNT100;
   1:  PR[91,1] = PR[90,1] + -19.706;
   1:  PR[91,2] = PR[90,2] + -16.511;
   1:  PR[91,3] = PR[90,3] + 9.133;
   1:L PR[91] R[100]mm/sec CNT100;
   1:  PR[91,1] = PR[90,1] + -18.854;
   1:  PR[91,2] = PR[90,2] + -16.482;
   1:  PR[91,3] = PR[90,3] + 9.138;
   1:L PR[91] R[100]mm/sec CNT100;
   1:  PR[91,1] = PR[90,1] + -18.033;
   1:  PR[91,2] = PR[90,2] + -16.414;
   1:  PR[91,3] = PR[90,3] + 9.143;
   1:L PR[91] R[100]mm/sec CNT100;
   1:  PR[91,1] = PR[90,1] + -17.205;
   1:  PR[91,2] = PR[90,2] + -16.305;
   1:  PR[91,3] = PR[90,3] + 9.149;
   1:L PR[91] R[100]mm/sec CNT100;
   1:  PR[91,1] = PR[90,1] + -16.387;
   1:  PR[91,2] = PR[90,2] + -16.156;
   1:  PR[91,3] = PR[90,3] + 9.154;
   1:L PR[91] R[100]mm/sec CNT100;
   1:  PR[91,1] = PR[90,1] + -15.380;
   1:  PR[91,2] = PR[90,2] + -15.915;
   1:  PR[91,3] = PR[90,3] + 9.159;
   1:L PR[91] R[100]mm/sec CNT100;
   1:  PR[91,1] = PR[90,1] + -14.772;
   1:  PR[91,2] = PR[90,2] + -15.740;
   1:  PR[91,3] = PR[90,3] + 9.165;
   1:L PR[91] R[100]mm/sec CNT100;
   1:  PR[91,1] = PR[90,1] + -13.983;
   1:  PR[91,2] = PR[90,2] + -15.475;
   1:  PR[91,3] = PR[90,3] + 9.169;
   1:L PR[91] R[100]mm/sec CNT100;
   1:  PR[91,1] = PR[90,1] + -13.207;
   1:  PR[91,2] = PR[90,2] + -15.171;
   1:  PR[91,3] = PR[90,3] + 9.174;
   1:L PR[91] R[100]mm/sec CNT100;
   1:  PR[91,1] = PR[90,1] + -12.899;
   1:  PR[91,2] = PR[90,2] + -15.035;
   1:  PR[91,3] = PR[90,3] + 9.179;
   1:L PR[91] R[100]mm/sec CNT100;
   1:  PR[91,1] = PR[90,1] + -12.451;
   1:  PR[91,2] = PR[90,2] + -14.832;
   1:  PR[91,3] = PR[90,3] + 9.181;
   1:L PR[91] R[100]mm/sec CNT100;
   1:  PR[91,1] = PR[90,1] + -11.710;
   1:  PR[91,2] = PR[90,2] + -14.455;
   1:  PR[91,3] = PR[90,3] + 9.184;
   1:L PR[91] R[100]mm/sec CNT100;
   1:  PR[91,1] = PR[90,1] + -10.987;
   1:  PR[91,2] = PR[90,2] + -14.043;
   1:  PR[91,3] = PR[90,3] + 9.189;
   1:L PR[91] R[100]mm/sec CNT100;
   1:  PR[91,1] = PR[90,1] + -10.576;
   1:  PR[91,2] = PR[90,2] + -13.786;
   1:  PR[91,3] = PR[90,3] + 9.194;
   1:L PR[91] R[100]mm/sec CNT100;
   1:  PR[91,1] = PR[90,1] + -10.291;
   1:  PR[91,2] = PR[90,2] + -13.601;
   1:  PR[91,3] = PR[90,3] + 9.197;
   1:L PR[91] R[100]mm/sec CNT100;
   1:  PR[91,1] = PR[90,1] + -9.612;
   1:  PR[91,2] = PR[90,2] + -13.122;
   1:  PR[91,3] = PR[90,3] + 9.199;
   1:L PR[91] R[100]mm/sec CNT100;
   1:  PR[91,1] = PR[90,1] + -8.960;
   1:  PR[91,2] = PR[90,2] + -12.613;
   1:  PR[91,3] = PR[90,3] + 9.204;
   1:L PR[91] R[100]mm/sec CNT100;
   1:  PR[91,1] = PR[90,1] + -8.333;
   1:  PR[91,2] = PR[90,2] + -12.072;
   1:  PR[91,3] = PR[90,3] + 9.209;
   1:L PR[91] R[100]mm/sec CNT100;
   1:  PR[91,1] = PR[90,1] + -7.848;
   1:  PR[91,2] = PR[90,2] + -11.614;
   1:  PR[91,3] = PR[90,3] + 9.215;
   1:L PR[91] R[100]mm/sec CNT100;
   1:  PR[91,1] = PR[90,1] + -7.162;
   1:  PR[91,2] = PR[90,2] + -10.904;
   1:  PR[91,3] = PR[90,3] + 9.219;
   1:L PR[91] R[100]mm/sec CNT100;
   1:  PR[91,1] = PR[90,1] + -6.622;
   1:  PR[91,2] = PR[90,2] + -10.281;
   1:  PR[91,3] = PR[90,3] + 9.225;
   1:L PR[91] R[100]mm/sec CNT100;
   1:  PR[91,1] = PR[90,1] + -6.113;
   1:  PR[91,2] = PR[90,2] + -9.630;
   1:  PR[91,3] = PR[90,3] + 9.230;
   1:L PR[91] R[100]mm/sec CNT100;
   1:  PR[91,1] = PR[90,1] + -5.632;
   1:  PR[91,2] = PR[90,2] + -8.951;
   1:  PR[91,3] = PR[90,3] + 9.235;
   1:L PR[91] R[100]mm/sec CNT100;
   1:  PR[91,1] = PR[90,1] + -5.178;
   1:  PR[91,2] = PR[90,2] + -8.237;
   1:  PR[91,3] = PR[90,3] + 9.240;
   1:L PR[91] R[100]mm/sec CNT100;
   1:  PR[91,1] = PR[90,1] + -4.759;
   1:  PR[91,2] = PR[90,2] + -7.501;
   1:  PR[91,3] = PR[90,3] + 9.245;
   1:L PR[91] R[100]mm/sec CNT100;
   1:  PR[91,1] = PR[90,1] + -4.378;
   1:  PR[91,2] = PR[90,2] + -6.746;
   1:  PR[91,3] = PR[90,3] + 9.250;
   1:L PR[91] R[100]mm/sec CNT100;
   1:  PR[91,1] = PR[90,1] + -4.090;
   1:  PR[91,2] = PR[90,2] + -6.102;
   1:  PR[91,3] = PR[90,3] + 9.255;
   1:L PR[91] R[100]mm/sec CNT100;
   1:  PR[91,1] = PR[90,1] + -3.732;
   1:  PR[91,2] = PR[90,2] + -5.191;
   1:  PR[91,3] = PR[90,3] + 9.260;
   1:L PR[91] R[100]mm/sec CNT100;
   1:  PR[91,1] = PR[90,1] + -3.470;
   1:  PR[91,2] = PR[90,2] + -4.398;
   1:  PR[91,3] = PR[90,3] + 9.266;
   1:L PR[91] R[100]mm/sec CNT100;
   1:  PR[91,1] = PR[90,1] + -3.247;
   1:  PR[91,2] = PR[90,2] + -3.592;
   1:  PR[91,3] = PR[90,3] + 9.271;
   1:L PR[91] R[100]mm/sec CNT100;
   1:  PR[91,1] = PR[90,1] + -3.073;
   1:  PR[91,2] = PR[90,2] + -2.820;
   1:  PR[91,3] = PR[90,3] + 9.276;
   1:L PR[91] R[100]mm/sec CNT100;
   1:  PR[91,1] = PR[90,1] + -2.959;
   1:  PR[91,2] = PR[90,2] + -2.426;
   1:  PR[91,3] = PR[90,3] + 9.281;
   1:L PR[91] R[100]mm/sec CNT100;
   1:  PR[91,1] = PR[90,1] + -2.827;
   1:  PR[91,2] = PR[90,2] + -2.086;
   1:  PR[91,3] = PR[90,3] + 9.283;
   1:L PR[91] R[100]mm/sec CNT100;
   1:  PR[91,1] = PR[90,1] + -2.679;
   1:  PR[91,2] = PR[90,2] + -1.777;
   1:  PR[91,3] = PR[90,3] + 9.285;
   1:L PR[91] R[100]mm/sec CNT100;
   1:  PR[91,1] = PR[90,1] + -2.515;
   1:  PR[91,2] = PR[90,2] + -1.507;
   1:  PR[91,3] = PR[90,3] + 9.288;
   1:L PR[91] R[100]mm/sec CNT100;
   1:  PR[91,1] = PR[90,1] + -2.274;
   1:  PR[91,2] = PR[90,2] + -1.196;
   1:  PR[91,3] = PR[90,3] + 9.289;
   1:L PR[91] R[100]mm/sec CNT100;
   1:  PR[91,1] = PR[90,1] + -1.916;
   1:  PR[91,2] = PR[90,2] + -0.843;
   1:  PR[91,3] = PR[90,3] + 9.292;
   1:L PR[91] R[100]mm/sec CNT100;
   1:  PR[91,1] = PR[90,1] + -1.631;
   1:  PR[91,2] = PR[90,2] + -0.641;
   1:  PR[91,3] = PR[90,3] + 9.295;
   1:L PR[91] R[100]mm/sec CNT100;
   1:  PR[91,1] = PR[90,1] + -1.326;
   1:  PR[91,2] = PR[90,2] + -0.485;
   1:  PR[91,3] = PR[90,3] + 9.297;
   1:L PR[91] R[100]mm/sec CNT100;
   1:  PR[91,1] = PR[90,1] + -0.911;
   1:  PR[91,2] = PR[90,2] + -0.314;
   1:  PR[91,3] = PR[90,3] + 9.299;
   1:L PR[91] R[100]mm/sec CNT100;
   1:  PR[91,1] = PR[90,1] + -0.229;
   1:  PR[91,2] = PR[90,2] + -0.209;
   1:  PR[91,3] = PR[90,3] + 9.302;
   1:L PR[91] R[100]mm/sec CNT100;
   1:  PR[91,1] = PR[90,1] + 0.404;
   1:  PR[91,2] = PR[90,2] + -0.258;
   1:  PR[91,3] = PR[90,3] + 9.306;
   1:L PR[91] R[100]mm/sec CNT100;
   1:  PR[91] = PR[90];
   1:  PR[91,1] = PR[90,1] + 0.727;
   1:  PR[91,2] = PR[90,2] + -1.413;
   1:  PR[91,3] = PR[90,3] + 10.640;
   1:L PR[91] R[100]mm/sec CNT100;
   1:  PR[91,1] = PR[90,1] + 1.096;
   1:  PR[91,2] = PR[90,2] + -1.579;
   1:  PR[91,3] = PR[90,3] + 9.313;
   1:L PR[91] R[100]mm/sec CNT100;
   1:  PR[91,1] = PR[90,1] + 1.449;
   1:  PR[91,2] = PR[90,2] + -1.805;
   1:  PR[91,3] = PR[90,3] + 9.315;
   1:L PR[91] R[100]mm/sec CNT100;
   1:  PR[91,1] = PR[90,1] + 1.785;
   1:  PR[91,2] = PR[90,2] + -2.097;
   1:  PR[91,3] = PR[90,3] + 9.318;
   1:L PR[91] R[100]mm/sec CNT100;
   1:  PR[91,1] = PR[90,1] + 2.059;
   1:  PR[91,2] = PR[90,2] + -2.402;
   1:  PR[91,3] = PR[90,3] + 9.321;
   1:L PR[91] R[100]mm/sec CNT100;
   1:  PR[91,1] = PR[90,1] + 2.301;
   1:  PR[91,2] = PR[90,2] + -2.743;
   1:  PR[91,3] = PR[90,3] + 9.323;
   1:L PR[91] R[100]mm/sec CNT100;
   1:  PR[91,1] = PR[90,1] + 2.507;
   1:  PR[91,2] = PR[90,2] + -3.112;
   1:  PR[91,3] = PR[90,3] + 9.326;
   1:L PR[91] R[100]mm/sec CNT100;
   1:  PR[91,1] = PR[90,1] + 2.678;
   1:  PR[91,2] = PR[90,2] + -3.508;
   1:  PR[91,3] = PR[90,3] + 9.329;
   1:L PR[91] R[100]mm/sec CNT100;
   1:  PR[91,1] = PR[90,1] + 3.112;
   1:  PR[91,2] = PR[90,2] + -4.911;
   1:  PR[91,3] = PR[90,3] + 9.331;
   1:L PR[91] R[100]mm/sec CNT100;
   1:  PR[91,1] = PR[90,1] + 3.402;
   1:  PR[91,2] = PR[90,2] + -5.695;
   1:  PR[91,3] = PR[90,3] + 9.340;
   1:L PR[91] R[100]mm/sec CNT100;
   1:  PR[91,1] = PR[90,1] + 3.734;
   1:  PR[91,2] = PR[90,2] + -6.470;
   1:  PR[91,3] = PR[90,3] + 9.346;
   1:L PR[91] R[100]mm/sec CNT100;
   1:  PR[91,1] = PR[90,1] + 3.952;
   1:  PR[91,2] = PR[90,2] + -6.925;
   1:  PR[91,3] = PR[90,3] + 9.351;
   1:L PR[91] R[100]mm/sec CNT100;
   1:  PR[91,1] = PR[90,1] + 4.329;
   1:  PR[91,2] = PR[90,2] + -7.647;
   1:  PR[91,3] = PR[90,3] + 9.354;
   1:L PR[91] R[100]mm/sec CNT100;
   1:  PR[91,1] = PR[90,1] + 4.737;
   1:  PR[91,2] = PR[90,2] + -8.348;
   1:  PR[91,3] = PR[90,3] + 9.359;
   1:L PR[91] R[100]mm/sec CNT100;
   1:  PR[91,1] = PR[90,1] + 5.179;
   1:  PR[91,2] = PR[90,2] + -9.029;
   1:  PR[91,3] = PR[90,3] + 9.364;
   1:L PR[91] R[100]mm/sec CNT100;
   1:  PR[91,1] = PR[90,1] + 5.654;
   1:  PR[91,2] = PR[90,2] + -9.692;
   1:  PR[91,3] = PR[90,3] + 9.369;
   1:L PR[91] R[100]mm/sec CNT100;
   1:  PR[91,1] = PR[90,1] + 5.970;
   1:  PR[91,2] = PR[90,2] + -10.100;
   1:  PR[91,3] = PR[90,3] + 9.374;
   1:L PR[91] R[100]mm/sec CNT100;
   1:  PR[91,1] = PR[90,1] + 6.529;
   1:  PR[91,2] = PR[90,2] + -10.761;
   1:  PR[91,3] = PR[90,3] + 9.377;
   1:L PR[91] R[100]mm/sec CNT100;
   1:  PR[91,1] = PR[90,1] + 7.122;
   1:  PR[91,2] = PR[90,2] + -11.392;
   1:  PR[91,3] = PR[90,3] + 9.383;
   1:L PR[91] R[100]mm/sec CNT100;
   1:  PR[91,1] = PR[90,1] + 7.746;
   1:  PR[91,2] = PR[90,2] + -11.993;
   1:  PR[91,3] = PR[90,3] + 9.388;
   1:L PR[91] R[100]mm/sec CNT100;
   1:  PR[91,1] = PR[90,1] + 8.459;
   1:  PR[91,2] = PR[90,2] + -12.609;
   1:  PR[91,3] = PR[90,3] + 9.394;
   1:L PR[91] R[100]mm/sec CNT100;
   1:  PR[91,1] = PR[90,1] + 9.100;
   1:  PR[91,2] = PR[90,2] + -13.109;
   1:  PR[91,3] = PR[90,3] + 9.399;
   1:L PR[91] R[100]mm/sec CNT100;
   1:  PR[91,1] = PR[90,1] + 9.794;
   1:  PR[91,2] = PR[90,2] + -13.599;
   1:  PR[91,3] = PR[90,3] + 9.405;
   1:L PR[91] R[100]mm/sec CNT100;
   1:  PR[91,1] = PR[90,1] + 10.518;
   1:  PR[91,2] = PR[90,2] + -14.059;
   1:  PR[91,3] = PR[90,3] + 9.410;
   1:L PR[91] R[100]mm/sec CNT100;
   1:  PR[91,1] = PR[90,1] + 11.264;
   1:  PR[91,2] = PR[90,2] + -14.482;
   1:  PR[91,3] = PR[90,3] + 9.415;
   1:L PR[91] R[100]mm/sec CNT100;
   1:  PR[91,1] = PR[90,1] + 12.030;
   1:  PR[91,2] = PR[90,2] + -14.868;
   1:  PR[91,3] = PR[90,3] + 9.420;
   1:L PR[91] R[100]mm/sec CNT100;
   1:  PR[91,1] = PR[90,1] + 12.813;
   1:  PR[91,2] = PR[90,2] + -15.215;
   1:  PR[91,3] = PR[90,3] + 9.426;
   1:L PR[91] R[100]mm/sec CNT100;
   1:  PR[91,1] = PR[90,1] + 13.612;
   1:  PR[91,2] = PR[90,2] + -15.523;
   1:  PR[91,3] = PR[90,3] + 9.431;
   1:L PR[91] R[100]mm/sec CNT100;
   1:  PR[91,1] = PR[90,1] + 14.424;
   1:  PR[91,2] = PR[90,2] + -15.791;
   1:  PR[91,3] = PR[90,3] + 9.436;
   1:L PR[91] R[100]mm/sec CNT100;
   1:  PR[91,1] = PR[90,1] + 15.249;
   1:  PR[91,2] = PR[90,2] + -16.019;
   1:  PR[91,3] = PR[90,3] + 9.442;
   1:L PR[91] R[100]mm/sec CNT100;
   1:  PR[91,1] = PR[90,1] + 16.082;
   1:  PR[91,2] = PR[90,2] + -16.206;
   1:  PR[91,3] = PR[90,3] + 9.447;
   1:L PR[91] R[100]mm/sec CNT100;
   1:  PR[91,1] = PR[90,1] + 16.923;
   1:  PR[91,2] = PR[90,2] + -16.352;
   1:  PR[91,3] = PR[90,3] + 9.452;
   1:L PR[91] R[100]mm/sec CNT100;
   1:  PR[91,1] = PR[90,1] + 17.770;
   1:  PR[91,2] = PR[90,2] + -16.456;
   1:  PR[91,3] = PR[90,3] + 9.458;
   1:L PR[91] R[100]mm/sec CNT100;
   1:  PR[91,1] = PR[90,1] + 18.619;
   1:  PR[91,2] = PR[90,2] + -16.518;
   1:  PR[91,3] = PR[90,3] + 9.463;
   1:L PR[91] R[100]mm/sec CNT100;
   1:  PR[91,1] = PR[90,1] + 19.470;
   1:  PR[91,2] = PR[90,2] + -16.538;
   1:  PR[91,3] = PR[90,3] + 9.468;
   1:L PR[91] R[100]mm/sec CNT100;
   1:  PR[91,1] = PR[90,1] + 20.340;
   1:  PR[91,2] = PR[90,2] + -16.516;
   1:  PR[91,3] = PR[90,3] + 9.474;
   1:L PR[91] R[100]mm/sec CNT100;
   1:  PR[91,1] = PR[90,1] + 21.157;
   1:  PR[91,2] = PR[90,2] + -16.455;
   1:  PR[91,3] = PR[90,3] + 9.479;
   1:L PR[91] R[100]mm/sec CNT100;
   1:  PR[91,1] = PR[90,1] + 21.983;
   1:  PR[91,2] = PR[90,2] + -16.354;
   1:  PR[91,3] = PR[90,3] + 9.484;
   1:L PR[91] R[100]mm/sec CNT100;
   1:  PR[91,1] = PR[90,1] + 22.803;
   1:  PR[91,2] = PR[90,2] + -16.213;
   1:  PR[91,3] = PR[90,3] + 9.489;
   1:L PR[91] R[100]mm/sec CNT100;
   1:  PR[91,1] = PR[90,1] + 23.617;
   1:  PR[91,2] = PR[90,2] + -16.032;
   1:  PR[91,3] = PR[90,3] + 9.494;
   1:L PR[91] R[100]mm/sec CNT100;
   1:  PR[91,1] = PR[90,1] + 24.421;
   1:  PR[91,2] = PR[90,2] + -15.812;
   1:  PR[91,3] = PR[90,3] + 9.500;
   1:L PR[91] R[100]mm/sec CNT100;
   1:  PR[91,1] = PR[90,1] + 25.214;
   1:  PR[91,2] = PR[90,2] + -15.554;
   1:  PR[91,3] = PR[90,3] + 9.505;
   1:L PR[91] R[100]mm/sec CNT100;
   1:  PR[91,1] = PR[90,1] + 25.994;
   1:  PR[91,2] = PR[90,2] + -15.257;
   1:  PR[91,3] = PR[90,3] + 9.510;
   1:L PR[91] R[100]mm/sec CNT100;
   1:  PR[91,1] = PR[90,1] + 26.759;
   1:  PR[91,2] = PR[90,2] + -14.922;
   1:  PR[91,3] = PR[90,3] + 9.515;
   1:L PR[91] R[100]mm/sec CNT100;
   1:  PR[91,1] = PR[90,1] + 27.507;
   1:  PR[91,2] = PR[90,2] + -14.551;
   1:  PR[91,3] = PR[90,3] + 9.520;
   1:L PR[91] R[100]mm/sec CNT100;
   1:  PR[91,1] = PR[90,1] + 28.236;
   1:  PR[91,2] = PR[90,2] + -14.143;
   1:  PR[91,3] = PR[90,3] + 9.526;
   1:L PR[91] R[100]mm/sec CNT100;
   1:  PR[91,1] = PR[90,1] + 28.945;
   1:  PR[91,2] = PR[90,2] + -13.701;
   1:  PR[91,3] = PR[90,3] + 9.531;
   1:L PR[91] R[100]mm/sec CNT100;
   1:  PR[91,1] = PR[90,1] + 29.631;
   1:  PR[91,2] = PR[90,2] + -13.224;
   1:  PR[91,3] = PR[90,3] + 9.536;
   1:L PR[91] R[100]mm/sec CNT100;
   1:  PR[91,1] = PR[90,1] + 30.293;
   1:  PR[91,2] = PR[90,2] + -12.714;
   1:  PR[91,3] = PR[90,3] + 9.541;
   1:L PR[91] R[100]mm/sec CNT100;
   1:  PR[91,1] = PR[90,1] + 30.929;
   1:  PR[91,2] = PR[90,2] + -12.172;
   1:  PR[91,3] = PR[90,3] + 9.546;
   1:L PR[91] R[100]mm/sec CNT100;
   1:  PR[91,1] = PR[90,1] + 31.538;
   1:  PR[91,2] = PR[90,2] + -11.599;
   1:  PR[91,3] = PR[90,3] + 9.552;
   1:L PR[91] R[100]mm/sec CNT100;
   1:  PR[91,1] = PR[90,1] + 32.118;
   1:  PR[91,2] = PR[90,2] + -10.997;
   1:  PR[91,3] = PR[90,3] + 9.557;
   1:L PR[91] R[100]mm/sec CNT100;
   1:  PR[91,1] = PR[90,1] + 32.668;
   1:  PR[91,2] = PR[90,2] + -10.367;
   1:  PR[91,3] = PR[90,3] + 9.562;
   1:L PR[91] R[100]mm/sec CNT100;
   1:  PR[91,1] = PR[90,1] + 33.187;
   1:  PR[91,2] = PR[90,2] + -9.709;
   1:  PR[91,3] = PR[90,3] + 9.567;
   1:L PR[91] R[100]mm/sec CNT100;
   1:  PR[91,1] = PR[90,1] + 33.672;
   1:  PR[91,2] = PR[90,2] + -9.027;
   1:  PR[91,3] = PR[90,3] + 9.572;
   1:L PR[91] R[100]mm/sec CNT100;
   1:  PR[91,1] = PR[90,1] + 34.124;
   1:  PR[91,2] = PR[90,2] + -8.321;
   1:  PR[91,3] = PR[90,3] + 9.578;
   1:L PR[91] R[100]mm/sec CNT100;
   1:  PR[91,1] = PR[90,1] + 34.540;
   1:  PR[91,2] = PR[90,2] + -7.595;
   1:  PR[91,3] = PR[90,3] + 9.583;
   1:L PR[91] R[100]mm/sec CNT100;
   1:  PR[91,1] = PR[90,1] + 34.920;
   1:  PR[91,2] = PR[90,2] + -6.850;
   1:  PR[91,3] = PR[90,3] + 9.588;
   1:L PR[91] R[100]mm/sec CNT100;
   1:  PR[91,1] = PR[90,1] + 35.262;
   1:  PR[91,2] = PR[90,2] + -6.087;
   1:  PR[91,3] = PR[90,3] + 9.593;
   1:L PR[91] R[100]mm/sec CNT100;
   1:  PR[91,1] = PR[90,1] + 35.566;
   1:  PR[91,2] = PR[90,2] + -5.311;
   1:  PR[91,3] = PR[90,3] + 9.598;
   1:L PR[91] R[100]mm/sec CNT100;
   1:  PR[91,1] = PR[90,1] + 35.831;
   1:  PR[91,2] = PR[90,2] + -4.521;
   1:  PR[91,3] = PR[90,3] + 9.604;
   1:L PR[91] R[100]mm/sec CNT100;
   1:  PR[91,1] = PR[90,1] + 36.057;
   1:  PR[91,2] = PR[90,2] + -3.721;
   1:  PR[91,3] = PR[90,3] + 9.609;
   1:L PR[91] R[100]mm/sec CNT100;
   1:  PR[91,1] = PR[90,1] + 36.242;
   1:  PR[91,2] = PR[90,2] + -2.909;
   1:  PR[91,3] = PR[90,3] + 9.614;
   1:L PR[91] R[100]mm/sec CNT100;
   1:  PR[91,1] = PR[90,1] + 36.386;
   1:  PR[91,2] = PR[90,2] + -2.088;
   1:  PR[91,3] = PR[90,3] + 9.619;
   1:L PR[91] R[100]mm/sec CNT100;
   1:  PR[91,1] = PR[90,1] + 36.490;
   1:  PR[91,2] = PR[90,2] + -1.257;
   1:  PR[91,3] = PR[90,3] + 9.624;
   1:L PR[91] R[100]mm/sec CNT100;
   1:  PR[91,1] = PR[90,1] + 36.552;
   1:  PR[91,2] = PR[90,2] + -0.418;
   1:  PR[91,3] = PR[90,3] + 9.630;
   1:L PR[91] R[100]mm/sec CNT100;
   1:  PR[91,1] = PR[90,1] + 36.573;
   1:  PR[91,2] = PR[90,2] + 0.428;
   1:  PR[91,3] = PR[90,3] + 9.635;
   1:L PR[91] R[100]mm/sec CNT100;
   1:  PR[91,1] = PR[90,1] + 36.552;
   1:  PR[91,2] = PR[90,2] + 1.274;
   1:  PR[91,3] = PR[90,3] + 9.640;
   1:L PR[91] R[100]mm/sec CNT100;
   1:  PR[91,1] = PR[90,1] + 36.490;
   1:  PR[91,2] = PR[90,2] + 2.112;
   1:  PR[91,3] = PR[90,3] + 9.645;
   1:L PR[91] R[100]mm/sec CNT100;
   1:  PR[91,1] = PR[90,1] + 36.386;
   1:  PR[91,2] = PR[90,2] + 2.943;
   1:  PR[91,3] = PR[90,3] + 9.651;
   1:L PR[91] R[100]mm/sec CNT100;
   1:  PR[91,1] = PR[90,1] + 36.242;
   1:  PR[91,2] = PR[90,2] + 3.764;
   1:  PR[91,3] = PR[90,3] + 9.656;
   1:L PR[91] R[100]mm/sec CNT100;
   1:  PR[91,1] = PR[90,1] + 36.057;
   1:  PR[91,2] = PR[90,2] + 4.576;
   1:  PR[91,3] = PR[90,3] + 9.661;
   1:L PR[91] R[100]mm/sec CNT100;
   1:  PR[91,1] = PR[90,1] + 35.831;
   1:  PR[91,2] = PR[90,2] + 5.377;
   1:  PR[91,3] = PR[90,3] + 9.666;
   1:L PR[91] R[100]mm/sec CNT100;
   1:  PR[91,1] = PR[90,1] + 35.566;
   1:  PR[91,2] = PR[90,2] + 6.166;
   1:  PR[91,3] = PR[90,3] + 9.671;
   1:L PR[91] R[100]mm/sec CNT100;
   1:  PR[91,1] = PR[90,1] + 35.262;
   1:  PR[91,2] = PR[90,2] + 6.943;
   1:  PR[91,3] = PR[90,3] + 9.676;
   1:L PR[91] R[100]mm/sec CNT100;
   1:  PR[91,1] = PR[90,1] + 34.920;
   1:  PR[91,2] = PR[90,2] + 7.705;
   1:  PR[91,3] = PR[90,3] + 9.682;
   1:L PR[91] R[100]mm/sec CNT100;
   1:  PR[91,1] = PR[90,1] + 34.540;
   1:  PR[91,2] = PR[90,2] + 8.450;
   1:  PR[91,3] = PR[90,3] + 9.687;
   1:L PR[91] R[100]mm/sec CNT100;
   1:  PR[91,1] = PR[90,1] + 34.124;
   1:  PR[91,2] = PR[90,2] + 9.177;
   1:  PR[91,3] = PR[90,3] + 9.692;
   1:L PR[91] R[100]mm/sec CNT100;
   1:  PR[91,1] = PR[90,1] + 33.672;
   1:  PR[91,2] = PR[90,2] + 9.882;
   1:  PR[91,3] = PR[90,3] + 9.697;
   1:L PR[91] R[100]mm/sec CNT100;
   1:  PR[91,1] = PR[90,1] + 33.187;
   1:  PR[91,2] = PR[90,2] + 10.564;
   1:  PR[91,3] = PR[90,3] + 9.702;
   1:L PR[91] R[100]mm/sec CNT100;
   1:  PR[91,1] = PR[90,1] + 32.668;
   1:  PR[91,2] = PR[90,2] + 11.222;
   1:  PR[91,3] = PR[90,3] + 9.708;
   1:L PR[91] R[100]mm/sec CNT100;
   1:  PR[91,1] = PR[90,1] + 32.118;
   1:  PR[91,2] = PR[90,2] + 11.852;
   1:  PR[91,3] = PR[90,3] + 9.713;
   1:L PR[91] R[100]mm/sec CNT100;
   1:  PR[91,1] = PR[90,1] + 31.538;
   1:  PR[91,2] = PR[90,2] + 12.455;
   1:  PR[91,3] = PR[90,3] + 9.718;
   1:L PR[91] R[100]mm/sec CNT100;
   1:  PR[91,1] = PR[90,1] + 30.929;
   1:  PR[91,2] = PR[90,2] + 13.027;
   1:  PR[91,3] = PR[90,3] + 9.723;
   1:L PR[91] R[100]mm/sec CNT100;
   1:  PR[91,1] = PR[90,1] + 30.293;
   1:  PR[91,2] = PR[90,2] + 13.569;
   1:  PR[91,3] = PR[90,3] + 9.728;
   1:L PR[91] R[100]mm/sec CNT100;
   1:  PR[91,1] = PR[90,1] + 29.630;
   1:  PR[91,2] = PR[90,2] + 14.080;
   1:  PR[91,3] = PR[90,3] + 9.734;
   1:L PR[91] R[100]mm/sec CNT100;
   1:  PR[91,1] = PR[90,1] + 29.330;
   1:  PR[91,2] = PR[90,2] + 14.289;
   1:  PR[91,3] = PR[90,3] + 9.739;
   1:L PR[91] R[100]mm/sec CNT100;
   1:  PR[91,1] = PR[90,1] + 28.945;
   1:  PR[91,2] = PR[90,2] + 14.555;
   1:  PR[91,3] = PR[90,3] + 9.741;
   1:L PR[91] R[100]mm/sec CNT100;
   1:  PR[91,1] = PR[90,1] + 28.236;
   1:  PR[91,2] = PR[90,2] + 14.998;
   1:  PR[91,3] = PR[90,3] + 9.744;
   1:L PR[91] R[100]mm/sec CNT100;
   1:  PR[91,1] = PR[90,1] + 27.506;
   1:  PR[91,2] = PR[90,2] + 15.406;
   1:  PR[91,3] = PR[90,3] + 9.749;
   1:L PR[91] R[100]mm/sec CNT100;
   1:  PR[91,1] = PR[90,1] + 27.077;
   1:  PR[91,2] = PR[90,2] + 15.621;
   1:  PR[91,3] = PR[90,3] + 9.754;
   1:L PR[91] R[100]mm/sec CNT100;
   1:  PR[91,1] = PR[90,1] + 26.760;
   1:  PR[91,2] = PR[90,2] + 15.777;
   1:  PR[91,3] = PR[90,3] + 9.757;
   1:L PR[91] R[100]mm/sec CNT100;
   1:  PR[91,1] = PR[90,1] + 25.994;
   1:  PR[91,2] = PR[90,2] + 16.112;
   1:  PR[91,3] = PR[90,3] + 9.760;
   1:L PR[91] R[100]mm/sec CNT100;
   1:  PR[91,1] = PR[90,1] + 25.214;
   1:  PR[91,2] = PR[90,2] + 16.409;
   1:  PR[91,3] = PR[90,3] + 9.765;
   1:L PR[91] R[100]mm/sec CNT100;
   1:  PR[91,1] = PR[90,1] + 24.643;
   1:  PR[91,2] = PR[90,2] + 16.597;
   1:  PR[91,3] = PR[90,3] + 9.770;
   1:L PR[91] R[100]mm/sec CNT100;
   1:  PR[91,1] = PR[90,1] + 23.614;
   1:  PR[91,2] = PR[90,2] + 16.888;
   1:  PR[91,3] = PR[90,3] + 9.774;
   1:L PR[91] R[100]mm/sec CNT100;
   1:  PR[91,1] = PR[90,1] + 22.804;
   1:  PR[91,2] = PR[90,2] + 17.068;
   1:  PR[91,3] = PR[90,3] + 9.780;
   1:L PR[91] R[100]mm/sec CNT100;
   1:  PR[91,1] = PR[90,1] + 21.983;
   1:  PR[91,2] = PR[90,2] + 17.209;
   1:  PR[91,3] = PR[90,3] + 9.786;
   1:L PR[91] R[100]mm/sec CNT100;
   1:  PR[91,1] = PR[90,1] + 21.157;
   1:  PR[91,2] = PR[90,2] + 17.311;
   1:  PR[91,3] = PR[90,3] + 9.791;
   1:L PR[91] R[100]mm/sec CNT100;
   1:  PR[91,1] = PR[90,1] + 20.320;
   1:  PR[91,2] = PR[90,2] + 17.372;
   1:  PR[91,3] = PR[90,3] + 9.796;
   1:L PR[91] R[100]mm/sec CNT100;
   1:  PR[91,1] = PR[90,1] + 19.470;
   1:  PR[91,2] = PR[90,2] + 17.393;
   1:  PR[91,3] = PR[90,3] + 9.801;
   1:L PR[91] R[100]mm/sec CNT100;
   1:  PR[91,1] = PR[90,1] + 18.619;
   1:  PR[91,2] = PR[90,2] + 17.373;
   1:  PR[91,3] = PR[90,3] + 9.806;
   1:L PR[91] R[100]mm/sec CNT100;
   1:  PR[91,1] = PR[90,1] + 17.770;
   1:  PR[91,2] = PR[90,2] + 17.311;
   1:  PR[91,3] = PR[90,3] + 9.812;
   1:L PR[91] R[100]mm/sec CNT100;
   1:  PR[91,1] = PR[90,1] + 16.923;
   1:  PR[91,2] = PR[90,2] + 17.207;
   1:  PR[91,3] = PR[90,3] + 9.817;
   1:L PR[91] R[100]mm/sec CNT100;
   1:  PR[91,1] = PR[90,1] + 16.082;
   1:  PR[91,2] = PR[90,2] + 17.061;
   1:  PR[91,3] = PR[90,3] + 9.822;
   1:L PR[91] R[100]mm/sec CNT100;
   1:  PR[91,1] = PR[90,1] + 15.249;
   1:  PR[91,2] = PR[90,2] + 16.874;
   1:  PR[91,3] = PR[90,3] + 9.828;
   1:L PR[91] R[100]mm/sec CNT100;
   1:  PR[91,1] = PR[90,1] + 14.424;
   1:  PR[91,2] = PR[90,2] + 16.646;
   1:  PR[91,3] = PR[90,3] + 9.833;
   1:L PR[91] R[100]mm/sec CNT100;
   1:  PR[91,1] = PR[90,1] + 13.612;
   1:  PR[91,2] = PR[90,2] + 16.378;
   1:  PR[91,3] = PR[90,3] + 9.838;
   1:L PR[91] R[100]mm/sec CNT100;
   1:  PR[91,1] = PR[90,1] + 12.813;
   1:  PR[91,2] = PR[90,2] + 16.070;
   1:  PR[91,3] = PR[90,3] + 9.844;
   1:L PR[91] R[100]mm/sec CNT100;
   1:  PR[91,1] = PR[90,1] + 12.030;
   1:  PR[91,2] = PR[90,2] + 15.723;
   1:  PR[91,3] = PR[90,3] + 9.849;
   1:L PR[91] R[100]mm/sec CNT100;
   1:  PR[91,1] = PR[90,1] + 11.264;
   1:  PR[91,2] = PR[90,2] + 15.337;
   1:  PR[91,3] = PR[90,3] + 9.854;
   1:L PR[91] R[100]mm/sec CNT100;
   1:  PR[91,1] = PR[90,1] + 10.519;
   1:  PR[91,2] = PR[90,2] + 14.914;
   1:  PR[91,3] = PR[90,3] + 9.860;
   1:L PR[91] R[100]mm/sec CNT100;
   1:  PR[91,1] = PR[90,1] + 9.794;
   1:  PR[91,2] = PR[90,2] + 14.455;
   1:  PR[91,3] = PR[90,3] + 9.865;
   1:L PR[91] R[100]mm/sec CNT100;
   1:  PR[91,1] = PR[90,1] + 9.092;
   1:  PR[91,2] = PR[90,2] + 13.958;
   1:  PR[91,3] = PR[90,3] + 9.870;
   1:L PR[91] R[100]mm/sec CNT100;
   1:  PR[91,1] = PR[90,1] + 8.403;
   1:  PR[91,2] = PR[90,2] + 13.419;
   1:  PR[91,3] = PR[90,3] + 9.876;
   1:L PR[91] R[100]mm/sec CNT100;
   1:  PR[91,1] = PR[90,1] + 7.843;
   1:  PR[91,2] = PR[90,2] + 12.935;
   1:  PR[91,3] = PR[90,3] + 9.881;
   1:L PR[91] R[100]mm/sec CNT100;
   1:  PR[91,1] = PR[90,1] + 7.120;
   1:  PR[91,2] = PR[90,2] + 12.245;
   1:  PR[91,3] = PR[90,3] + 9.886;
   1:L PR[91] R[100]mm/sec CNT100;
   1:  PR[91,1] = PR[90,1] + 6.692;
   1:  PR[91,2] = PR[90,2] + 11.794;
   1:  PR[91,3] = PR[90,3] + 9.892;
   1:L PR[91] R[100]mm/sec CNT100;
   1:  PR[91,1] = PR[90,1] + 5.970;
   1:  PR[91,2] = PR[90,2] + 10.955;
   1:  PR[91,3] = PR[90,3] + 9.896;
   1:L PR[91] R[100]mm/sec CNT100;
   1:  PR[91,1] = PR[90,1] + 5.449;
   1:  PR[91,2] = PR[90,2] + 10.272;
   1:  PR[91,3] = PR[90,3] + 9.903;
   1:L PR[91] R[100]mm/sec CNT100;
   1:  PR[91,1] = PR[90,1] + 4.963;
   1:  PR[91,2] = PR[90,2] + 9.563;
   1:  PR[91,3] = PR[90,3] + 9.908;
   1:L PR[91] R[100]mm/sec CNT100;
   1:  PR[91,1] = PR[90,1] + 4.514;
   1:  PR[91,2] = PR[90,2] + 8.834;
   1:  PR[91,3] = PR[90,3] + 9.913;
   1:L PR[91] R[100]mm/sec CNT100;
   1:  PR[91,1] = PR[90,1] + 4.104;
   1:  PR[91,2] = PR[90,2] + 8.087;
   1:  PR[91,3] = PR[90,3] + 9.919;
   1:L PR[91] R[100]mm/sec CNT100;
   1:  PR[91,1] = PR[90,1] + 3.733;
   1:  PR[91,2] = PR[90,2] + 7.324;
   1:  PR[91,3] = PR[90,3] + 9.924;
   1:L PR[91] R[100]mm/sec CNT100;
   1:  PR[91,1] = PR[90,1] + 3.402;
   1:  PR[91,2] = PR[90,2] + 6.550;
   1:  PR[91,3] = PR[90,3] + 9.929;
   1:L PR[91] R[100]mm/sec CNT100;
   1:  PR[91,1] = PR[90,1] + 3.113;
   1:  PR[91,2] = PR[90,2] + 5.767;
   1:  PR[91,3] = PR[90,3] + 9.934;
   1:L PR[91] R[100]mm/sec CNT100;
   1:  PR[91,1] = PR[90,1] + 2.678;
   1:  PR[91,2] = PR[90,2] + 4.363;
   1:  PR[91,3] = PR[90,3] + 9.940;
   1:L PR[91] R[100]mm/sec CNT100;
   1:  PR[91,1] = PR[90,1] + 2.507;
   1:  PR[91,2] = PR[90,2] + 3.967;
   1:  PR[91,3] = PR[90,3] + 9.949;
   1:L PR[91] R[100]mm/sec CNT100;
   1:  PR[91,1] = PR[90,1] + 2.301;
   1:  PR[91,2] = PR[90,2] + 3.598;
   1:  PR[91,3] = PR[90,3] + 9.952;
   1:L PR[91] R[100]mm/sec CNT100;
   1:  PR[91,1] = PR[90,1] + 2.059;
   1:  PR[91,2] = PR[90,2] + 3.257;
   1:  PR[91,3] = PR[90,3] + 9.954;
   1:L PR[91] R[100]mm/sec CNT100;
   1:  PR[91,1] = PR[90,1] + 1.782;
   1:  PR[91,2] = PR[90,2] + 2.949;
   1:  PR[91,3] = PR[90,3] + 9.957;
   1:L PR[91] R[100]mm/sec CNT100;
   1:  PR[91,1] = PR[90,1] + 1.448;
   1:  PR[91,2] = PR[90,2] + 2.660;
   1:  PR[91,3] = PR[90,3] + 9.959;
   1:L PR[91] R[100]mm/sec CNT100;
   1:  PR[91,1] = PR[90,1] + 1.096;
   1:  PR[91,2] = PR[90,2] + 2.434;
   1:  PR[91,3] = PR[90,3] + 9.962;
   1:L PR[91] R[100]mm/sec CNT100;
   1:  PR[91,1] = PR[90,1] + 0.732;
   1:  PR[91,2] = PR[90,2] + 2.270;
   1:  PR[91,3] = PR[90,3] + 9.965;
   1:L PR[91] R[100]mm/sec CNT100;
   1:  PR[91,1] = PR[90,1] + 0.355;
   1:  PR[91,2] = PR[90,2] + 2.166;
   1:  PR[91,3] = PR[90,3] + 9.967;
   1:L PR[91] R[100]mm/sec CNT100;
   1:  PR[91,1] = PR[90,1] + -0.113;
   1:  PR[91,2] = PR[90,2] + 2.118;
   1:  PR[91,3] = PR[90,3] + 9.970;
   1:L PR[91] R[100]mm/sec CNT100;
   1:  PR[91,1] = PR[90,1] + -0.508;
   1:  PR[91,2] = PR[90,2] + 2.150;
   1:  PR[91,3] = PR[90,3] + 9.973;
   1:L PR[91] R[100]mm/sec CNT100;
   1:  PR[91,1] = PR[90,1] + -0.914;
   1:  PR[91,2] = PR[90,2] + 2.250;
   1:  PR[91,3] = PR[90,3] + 9.975;
   1:L PR[91] R[100]mm/sec CNT100;
   1:  PR[91,1] = PR[90,1] + -1.356;
   1:  PR[91,2] = PR[90,2] + 2.445;
   1:  PR[91,3] = PR[90,3] + 9.978;
   1:L PR[91] R[100]mm/sec CNT100;
   1:  PR[91,1] = PR[90,1] + -1.688;
   1:  PR[91,2] = PR[90,2] + 2.660;
   1:  PR[91,3] = PR[90,3] + 9.981;
   1:L PR[91] R[100]mm/sec CNT100;
   1:  PR[91,1] = PR[90,1] + -2.023;
   1:  PR[91,2] = PR[90,2] + 2.950;
   1:  PR[91,3] = PR[90,3] + 9.983;
   1:L PR[91] R[100]mm/sec CNT100;
   1:  PR[91,1] = PR[90,1] + -2.299;
   1:  PR[91,2] = PR[90,2] + 3.257;
   1:  PR[91,3] = PR[90,3] + 9.986;
   1:L PR[91] R[100]mm/sec CNT100;
   1:  PR[91,1] = PR[90,1] + -2.541;
   1:  PR[91,2] = PR[90,2] + 3.598;
   1:  PR[91,3] = PR[90,3] + 9.988;
   1:L PR[91] R[100]mm/sec CNT100;
   1:  PR[91,1] = PR[90,1] + -2.747;
   1:  PR[91,2] = PR[90,2] + 3.967;
   1:  PR[91,3] = PR[90,3] + 9.991;
   1:L PR[91] R[100]mm/sec CNT100;
   1:  PR[91,1] = PR[90,1] + -2.919;
   1:  PR[91,2] = PR[90,2] + 4.363;
   1:  PR[91,3] = PR[90,3] + 9.994;
   1:L PR[91] R[100]mm/sec CNT100;
   1:  PR[91,1] = PR[90,1] + -3.353;
   1:  PR[91,2] = PR[90,2] + 5.768;
   1:  PR[91,3] = PR[90,3] + 9.996;
   1:L PR[91] R[100]mm/sec CNT100;
   1:  PR[91,1] = PR[90,1] + -3.644;
   1:  PR[91,2] = PR[90,2] + 6.553;
   1:  PR[91,3] = PR[90,3] + 10.005;
   1:L PR[91] R[100]mm/sec CNT100;
   1:  PR[91,1] = PR[90,1] + -3.975;
   1:  PR[91,2] = PR[90,2] + 7.330;
   1:  PR[91,3] = PR[90,3] + 10.011;
   1:L PR[91] R[100]mm/sec CNT100;
   1:  PR[91,1] = PR[90,1] + -4.346;
   1:  PR[91,2] = PR[90,2] + 8.094;
   1:  PR[91,3] = PR[90,3] + 10.016;
   1:L PR[91] R[100]mm/sec CNT100;
   1:  PR[91,1] = PR[90,1] + -4.756;
   1:  PR[91,2] = PR[90,2] + 8.843;
   1:  PR[91,3] = PR[90,3] + 10.021;
   1:L PR[91] R[100]mm/sec CNT100;
   1:  PR[91,1] = PR[90,1] + -5.205;
   1:  PR[91,2] = PR[90,2] + 9.572;
   1:  PR[91,3] = PR[90,3] + 10.026;
   1:L PR[91] R[100]mm/sec CNT100;
   1:  PR[91,1] = PR[90,1] + -5.690;
   1:  PR[91,2] = PR[90,2] + 10.280;
   1:  PR[91,3] = PR[90,3] + 10.032;
   1:L PR[91] R[100]mm/sec CNT100;
   1:  PR[91,1] = PR[90,1] + -6.211;
   1:  PR[91,2] = PR[90,2] + 10.962;
   1:  PR[91,3] = PR[90,3] + 10.037;
   1:L PR[91] R[100]mm/sec CNT100;
   1:  PR[91,1] = PR[90,1] + -6.934;
   1:  PR[91,2] = PR[90,2] + 11.798;
   1:  PR[91,3] = PR[90,3] + 10.042;
   1:L PR[91] R[100]mm/sec CNT100;
   1:  PR[91,1] = PR[90,1] + -7.362;
   1:  PR[91,2] = PR[90,2] + 12.250;
   1:  PR[91,3] = PR[90,3] + 10.049;
   1:L PR[91] R[100]mm/sec CNT100;
   1:  PR[91,1] = PR[90,1] + -7.989;
   1:  PR[91,2] = PR[90,2] + 12.851;
   1:  PR[91,3] = PR[90,3] + 10.053;
   1:L PR[91] R[100]mm/sec CNT100;
   1:  PR[91,1] = PR[90,1] + -8.700;
   1:  PR[91,2] = PR[90,2] + 13.466;
   1:  PR[91,3] = PR[90,3] + 10.059;
   1:L PR[91] R[100]mm/sec CNT100;
   1:  PR[91,1] = PR[90,1] + -9.342;
   1:  PR[91,2] = PR[90,2] + 13.965;
   1:  PR[91,3] = PR[90,3] + 10.064;
   1:L PR[91] R[100]mm/sec CNT100;
   1:  PR[91,1] = PR[90,1] + -10.037;
   1:  PR[91,2] = PR[90,2] + 14.456;
   1:  PR[91,3] = PR[90,3] + 10.070;
   1:L PR[91] R[100]mm/sec CNT100;
   1:  PR[91,1] = PR[90,1] + -10.760;
   1:  PR[91,2] = PR[90,2] + 14.915;
   1:  PR[91,3] = PR[90,3] + 10.075;
   1:L PR[91] R[100]mm/sec CNT100;
   1:  PR[91,1] = PR[90,1] + -11.506;
   1:  PR[91,2] = PR[90,2] + 15.339;
   1:  PR[91,3] = PR[90,3] + 10.080;
   1:L PR[91] R[100]mm/sec CNT100;
   1:  PR[91,1] = PR[90,1] + -12.272;
   1:  PR[91,2] = PR[90,2] + 15.724;
   1:  PR[91,3] = PR[90,3] + 10.085;
   1:L PR[91] R[100]mm/sec CNT100;
   1:  PR[91,1] = PR[90,1] + -13.055;
   1:  PR[91,2] = PR[90,2] + 16.072;
   1:  PR[91,3] = PR[90,3] + 10.091;
   1:L PR[91] R[100]mm/sec CNT100;
   1:  PR[91,1] = PR[90,1] + -13.853;
   1:  PR[91,2] = PR[90,2] + 16.380;
   1:  PR[91,3] = PR[90,3] + 10.096;
   1:L PR[91] R[100]mm/sec CNT100;
   1:  PR[91,1] = PR[90,1] + -14.666;
   1:  PR[91,2] = PR[90,2] + 16.648;
   1:  PR[91,3] = PR[90,3] + 10.101;
   1:L PR[91] R[100]mm/sec CNT100;
   1:  PR[91,1] = PR[90,1] + -15.490;
   1:  PR[91,2] = PR[90,2] + 16.875;
   1:  PR[91,3] = PR[90,3] + 10.107;
   1:L PR[91] R[100]mm/sec CNT100;
   1:  PR[91,1] = PR[90,1] + -16.323;
   1:  PR[91,2] = PR[90,2] + 17.062;
   1:  PR[91,3] = PR[90,3] + 10.112;
   1:L PR[91] R[100]mm/sec CNT100;
   1:  PR[91,1] = PR[90,1] + -17.164;
   1:  PR[91,2] = PR[90,2] + 17.207;
   1:  PR[91,3] = PR[90,3] + 10.117;
   1:L PR[91] R[100]mm/sec CNT100;
   1:  PR[91,1] = PR[90,1] + -18.010;
   1:  PR[91,2] = PR[90,2] + 17.311;
   1:  PR[91,3] = PR[90,3] + 10.123;
   1:L PR[91] R[100]mm/sec CNT100;
   1:  PR[91,1] = PR[90,1] + -18.860;
   1:  PR[91,2] = PR[90,2] + 17.373;
   1:  PR[91,3] = PR[90,3] + 10.128;
   1:L PR[91] R[100]mm/sec CNT100;
   1:  PR[91,1] = PR[90,1] + -19.710;
   1:  PR[91,2] = PR[90,2] + 17.393;
   1:  PR[91,3] = PR[90,3] + 10.133;
   1:L PR[91] R[100]mm/sec CNT100;
   1:  PR[91,1] = PR[90,1] + -20.580;
   1:  PR[91,2] = PR[90,2] + 17.371;
   1:  PR[91,3] = PR[90,3] + 10.139;
   1:L PR[91] R[100]mm/sec CNT100;
   1:  PR[91,1] = PR[90,1] + -21.397;
   1:  PR[91,2] = PR[90,2] + 17.310;
   1:  PR[91,3] = PR[90,3] + 10.144;
   1:L PR[91] R[100]mm/sec CNT100;
   1:  PR[91,1] = PR[90,1] + -22.223;
   1:  PR[91,2] = PR[90,2] + 17.209;
   1:  PR[91,3] = PR[90,3] + 10.149;
   1:L PR[91] R[100]mm/sec CNT100;
   1:  PR[91,1] = PR[90,1] + -23.043;
   1:  PR[91,2] = PR[90,2] + 17.068;
   1:  PR[91,3] = PR[90,3] + 10.154;
   1:L PR[91] R[100]mm/sec CNT100;
   1:  PR[91,1] = PR[90,1] + -23.854;
   1:  PR[91,2] = PR[90,2] + 16.888;
   1:  PR[91,3] = PR[90,3] + 10.159;
   1:L PR[91] R[100]mm/sec CNT100;
   1:  PR[91,1] = PR[90,1] + -24.882;
   1:  PR[91,2] = PR[90,2] + 16.597;
   1:  PR[91,3] = PR[90,3] + 10.165;
   1:L PR[91] R[100]mm/sec CNT100;
   1:  PR[91,1] = PR[90,1] + -25.453;
   1:  PR[91,2] = PR[90,2] + 16.409;
   1:  PR[91,3] = PR[90,3] + 10.171;
   1:L PR[91] R[100]mm/sec CNT100;
   1:  PR[91,1] = PR[90,1] + -26.234;
   1:  PR[91,2] = PR[90,2] + 16.112;
   1:  PR[91,3] = PR[90,3] + 10.175;
   1:L PR[91] R[100]mm/sec CNT100;
   1:  PR[91,1] = PR[90,1] + -26.998;
   1:  PR[91,2] = PR[90,2] + 15.777;
   1:  PR[91,3] = PR[90,3] + 10.180;
   1:L PR[91] R[100]mm/sec CNT100;
   1:  PR[91,1] = PR[90,1] + -27.746;
   1:  PR[91,2] = PR[90,2] + 15.405;
   1:  PR[91,3] = PR[90,3] + 10.185;
   1:L PR[91] R[100]mm/sec CNT100;
   1:  PR[91,1] = PR[90,1] + -28.476;
   1:  PR[91,2] = PR[90,2] + 14.997;
   1:  PR[91,3] = PR[90,3] + 10.191;
   1:L PR[91] R[100]mm/sec CNT100;
   1:  PR[91,1] = PR[90,1] + -28.843;
   1:  PR[91,2] = PR[90,2] + 14.769;
   1:  PR[91,3] = PR[90,3] + 10.196;
